C07315=1159.324,218.452,-63.263,-177.799,7.311,148.735
C07316=1159.328,218.203,-63.237,-177.801,7.309,148.735
C07317=1159.332,217.954,-63.212,-177.804,7.306,148.736
C07318=1159.336,217.706,-63.187,-177.807,7.304,148.736
C07319=1159.341,217.457,-63.161,-177.809,7.301,148.736
C07320=1159.346,217.208,-63.137,-177.812,7.300,148.736
C07321=1159.350,216.960,-63.111,-177.815,7.297,148.736
C07322=1159.354,216.711,-63.087,-177.818,7.294,148.737
C07323=1159.359,216.462,-63.061,-177.820,7.292,148.737
C07324=1159.364,216.214,-63.036,-177.823,7.289,148.737
C07325=1159.368,215.965,-63.011,-177.826,7.287,148.737
C07326=1159.372,215.716,-62.987,-177.828,7.284,148.737
C07327=1159.377,215.468,-62.961,-177.831,7.283,148.738
C07328=1159.382,215.219,-62.936,-177.834,7.280,148.738
C07329=1159.386,214.969,-62.911,-177.837,7.277,148.738
C07330=1159.390,214.722,-62.886,-177.839,7.275,148.738
C07331=1159.395,214.472,-62.861,-177.843,7.272,148.738
C07332=1159.400,214.224,-62.836,-177.845,7.270,148.739
C07333=1159.404,213.976,-62.812,-177.848,7.267,148.739
C07334=1159.409,213.726,-62.787,-177.850,7.266,148.739
C07335=1159.413,213.478,-62.761,-177.853,7.263,148.739
C07336=1159.417,213.229,-62.737,-177.856,7.261,148.739
C07337=1159.422,212.980,-62.712,-177.859,7.258,148.739
C07338=1159.427,212.732,-62.687,-177.862,7.255,148.740
C07339=1159.431,212.483,-62.662,-177.864,7.253,148.740
C07340=1159.435,212.234,-62.637,-177.867,7.251,148.740
C07341=1159.440,211.986,-62.612,-177.869,7.248,148.740
C07342=1159.445,211.737,-62.588,-177.873,7.246,148.741
C07343=1159.449,211.488,-62.563,-177.875,7.244,148.741
C07344=1159.454,211.239,-62.538,-177.878,7.241,148.741
C07345=1159.458,210.991,-62.513,-177.880,7.239,148.741
C07346=1159.463,210.742,-62.488,-177.883,7.236,148.741
C07347=1159.467,210.493,-62.464,-177.886,7.234,148.742
C07348=1159.472,210.223,-62.437,-177.889,7.232,148.742
C07349=1159.477,209.952,-62.411,-177.892,7.229,148.742
C07350=1159.482,209.681,-62.383,-177.895,7.226,148.742
C07351=1159.487,209.411,-62.357,-177.898,7.223,148.743
C07352=1159.492,209.163,-62.332,-177.901,7.222,148.743
C07353=1159.496,208.913,-62.308,-177.903,7.219,148.743
C07354=1159.501,208.665,-62.283,-177.906,7.217,148.743
C07355=1159.506,208.416,-62.258,-177.909,7.214,148.743
C07356=1159.510,208.167,-62.234,-177.911,7.212,148.744
C07357=1159.515,207.918,-62.209,-177.914,7.209,148.744
C07358=1159.519,207.670,-62.185,-177.917,7.207,148.744
C07359=1159.524,207.420,-62.160,-177.920,7.205,148.744
C07360=1159.528,207.172,-62.136,-177.922,7.203,148.745
C07361=1159.532,206.924,-62.111,-177.925,7.200,148.745
C07362=1159.537,206.675,-62.086,-177.928,7.198,148.745
C07363=1159.541,206.426,-62.062,-177.931,7.195,148.745
C07364=1159.546,206.178,-62.037,-177.933,7.193,148.746
C07365=1159.551,205.929,-62.014,-177.936,7.190,148.746
C07366=1159.556,205.679,-61.989,-177.939,7.189,148.746
C07367=1159.560,205.431,-61.965,-177.942,7.186,148.746
C07368=1159.565,205.182,-61.940,-177.944,7.184,148.746
C07369=1159.569,204.933,-61.916,-177.947,7.181,148.747
C07370=1159.573,204.684,-61.892,-177.950,7.179,148.747
C07371=1159.578,204.436,-61.867,-177.953,7.177,148.747
C07372=1159.583,204.187,-61.843,-177.955,7.175,148.747
C07373=1159.587,203.938,-61.819,-177.958,7.172,148.748
C07374=1159.592,203.689,-61.794,-177.961,7.170,148.748
C07375=1159.596,203.441,-61.770,-177.964,7.167,148.748
C07376=1159.601,203.192,-61.747,-177.966,7.165,148.748
C07377=1159.605,202.943,-61.721,-177.969,7.163,148.749
C07378=1159.610,202.694,-61.697,-177.971,7.161,148.749
C07379=1159.614,202.446,-61.673,-177.974,7.159,148.749
C07380=1159.619,202.197,-61.649,-177.977,7.156,148.749
C07381=1159.624,201.948,-61.625,-177.980,7.154,148.749
C07382=1159.628,201.699,-61.601,-177.983,7.151,148.750
C07383=1159.633,201.450,-61.576,-177.985,7.149,148.750
C07384=1159.637,201.202,-61.552,-177.988,7.147,148.750
C07385=1159.642,200.953,-61.529,-177.991,7.145,148.750
C07386=1159.646,200.704,-61.505,-177.994,7.142,148.751
C07387=1159.651,200.455,-61.480,-177.996,7.140,148.751
C07388=1159.655,200.207,-61.456,-177.999,7.137,148.751
C07389=1159.660,199.957,-61.432,-178.002,7.136,148.751
C07390=1159.664,199.709,-61.408,-178.005,7.133,148.752
C07391=1159.670,199.460,-61.383,-178.007,7.131,148.752
C07392=1159.674,199.211,-61.360,-178.010,7.129,148.752
C07393=1159.678,198.962,-61.336,-178.013,7.126,148.752
C07394=1159.682,198.714,-61.312,-178.015,7.124,148.753
C07395=1159.687,198.465,-61.288,-178.018,7.122,148.753
C07396=1159.692,198.216,-61.264,-178.021,7.120,148.753
C07397=1159.697,197.967,-61.240,-178.024,7.117,148.753
C07398=1159.701,197.719,-61.216,-178.026,7.115,148.754
C07399=1159.706,197.470,-61.193,-178.029,7.113,148.754
C07400=1159.710,197.221,-61.169,-178.032,7.110,148.754
C07401=1159.714,196.972,-61.144,-178.035,7.109,148.754
C07402=1159.719,196.723,-61.121,-178.037,7.106,148.755
C07403=1159.723,196.475,-61.097,-178.040,7.104,148.755
C07404=1159.729,196.225,-61.073,-178.043,7.101,148.755
C07405=1159.733,195.977,-61.049,-178.046,7.099,148.755
C07406=1159.738,195.728,-61.025,-178.048,7.098,148.756
C07407=1159.742,195.479,-61.001,-178.051,7.095,148.756
C07408=1159.747,195.230,-60.978,-178.054,7.093,148.756
C07409=1159.752,194.981,-60.955,-178.056,7.090,148.756
C07410=1159.756,194.733,-60.931,-178.059,7.088,148.757
C07411=1159.761,194.484,-60.907,-178.062,7.086,148.757
C07412=1159.765,194.235,-60.883,-178.065,7.083,148.757
C07413=1159.770,193.986,-60.860,-178.067,7.082,148.757
C07414=1159.774,193.737,-60.836,-178.071,7.079,148.758
C07415=1159.778,193.488,-60.812,-178.073,7.077,148.758
C07416=1159.783,193.239,-60.789,-178.075,7.075,148.758
C07417=1159.788,192.990,-60.765,-178.078,7.072,148.758
C07418=1159.792,192.742,-60.741,-178.081,7.071,148.759
C07419=1159.797,192.493,-60.718,-178.084,7.068,148.759
C07420=1159.802,192.244,-60.694,-178.086,7.066,148.759
C07421=1159.806,191.995,-60.670,-178.089,7.064,148.760
C07422=1159.811,191.746,-60.647,-178.092,7.062,148.760
C07423=1159.815,191.497,-60.624,-178.095,7.059,148.760
C07424=1159.820,191.249,-60.600,-178.098,7.057,148.760
C07425=1159.824,191.000,-60.576,-178.101,7.055,148.761
C07426=1159.829,190.751,-60.553,-178.103,7.053,148.761
C07427=1159.834,190.502,-60.530,-178.106,7.050,148.761
C07428=1159.839,190.253,-60.506,-178.109,7.049,148.762
C07429=1159.844,190.005,-60.482,-178.111,7.046,148.762
C07430=1159.848,189.756,-60.459,-178.114,7.044,148.762
C07431=1159.853,189.507,-60.436,-178.117,7.042,148.762
C07432=1159.858,189.258,-60.412,-178.120,7.039,148.762
C07433=1159.862,189.009,-60.389,-178.122,7.038,148.763
C07434=1159.866,188.760,-60.366,-178.125,7.036,148.763
C07435=1159.871,188.512,-60.342,-178.128,7.033,148.763
C07436=1159.875,188.263,-60.319,-178.130,7.031,148.764
C07437=1159.880,188.014,-60.295,-178.133,7.029,148.764
C07438=1159.885,187.765,-60.272,-178.136,7.026,148.764
C07439=1159.889,187.516,-60.249,-178.139,7.025,148.764
C07440=1159.893,187.267,-60.226,-178.142,7.022,148.765
C07441=1159.898,187.018,-60.203,-178.144,7.020,148.765
C07442=1159.903,186.769,-60.179,-178.147,7.018,148.765
C07443=1159.908,186.520,-60.156,-178.150,7.016,148.766
C07444=1159.913,186.271,-60.133,-178.152,7.014,148.766
C07445=1159.917,186.023,-60.110,-178.155,7.012,148.766
C07446=1159.922,185.774,-60.087,-178.158,7.009,148.766
C07447=1159.926,185.525,-60.063,-178.160,7.007,148.767
C07448=1159.931,185.276,-60.040,-178.163,7.005,148.767
C07449=1159.936,185.027,-60.017,-178.166,7.003,148.767
C07450=1159.940,184.778,-59.994,-178.169,7.001,148.767
C07451=1159.945,184.530,-59.971,-178.171,6.999,148.768
C07452=1159.950,184.260,-59.946,-178.175,6.996,148.768
C07453=1159.954,183.990,-59.921,-178.178,6.994,148.768
C07454=1159.959,183.720,-59.896,-178.180,6.992,148.769
C07455=1159.964,183.451,-59.870,-178.184,6.989,148.769
C07456=1159.969,183.202,-59.849,-178.186,6.987,148.769
C07457=1159.974,182.953,-59.825,-178.189,6.986,148.770
C07458=1159.979,182.704,-59.802,-178.192,6.983,148.770
C07459=1159.983,182.455,-59.779,-178.194,6.981,148.770
C07460=1159.987,182.206,-59.756,-178.197,6.979,148.771
C07461=1159.992,181.957,-59.732,-178.200,6.977,148.771
C07462=1159.997,181.709,-59.711,-178.203,6.975,148.771
C07463=1160.002,181.460,-59.687,-178.205,6.973,148.771
C07464=1160.006,181.211,-59.664,-178.208,6.970,148.772
C07465=1160.010,180.962,-59.641,-178.211,6.968,148.772
C07466=1160.015,180.713,-59.618,-178.214,6.967,148.772
C07467=1160.020,180.464,-59.596,-178.216,6.964,148.773
C07468=1160.025,180.215,-59.573,-178.219,6.962,148.773
C07469=1160.029,179.966,-59.550,-178.222,6.960,148.773
C07470=1160.034,179.717,-59.527,-178.224,6.958,148.774
C07471=1160.039,179.468,-59.504,-178.227,6.956,148.774
C07472=1160.043,179.220,-59.482,-178.230,6.954,148.774
C07473=1160.048,178.970,-59.459,-178.233,6.952,148.774
C07474=1160.052,178.721,-59.436,-178.236,6.950,148.775
C07475=1160.057,178.473,-59.413,-178.238,6.947,148.775
C07476=1160.062,178.223,-59.391,-178.241,6.946,148.775
C07477=1160.066,177.975,-59.368,-178.243,6.944,148.776
C07478=1160.071,177.726,-59.345,-178.247,6.941,148.776
C07479=1160.076,177.477,-59.323,-178.249,6.939,148.776
C07480=1160.080,177.228,-59.300,-178.252,6.937,148.777
C07481=1160.085,176.979,-59.277,-178.255,6.935,148.777
C07482=1160.090,176.730,-59.254,-178.258,6.933,148.777
C07483=1160.094,176.482,-59.232,-178.260,6.931,148.777
C07484=1160.099,176.232,-59.209,-178.263,6.929,148.778
C07485=1160.103,175.984,-59.187,-178.266,6.927,148.778
C07486=1160.108,175.734,-59.165,-178.268,6.925,148.778
C07487=1160.112,175.485,-59.141,-178.271,6.923,148.779
C07488=1160.117,175.237,-59.120,-178.274,6.920,148.779
C07489=1160.122,174.988,-59.096,-178.277,6.919,148.779
C07490=1160.126,174.738,-59.074,-178.279,6.917,148.780
C07491=1160.132,174.490,-59.051,-178.282,6.915,148.780
C07492=1160.136,174.241,-59.029,-178.285,6.912,148.780
C07493=1160.140,173.991,-59.007,-178.288,6.910,148.781
C07494=1160.145,173.743,-58.984,-178.290,6.909,148.781
C07495=1160.150,173.494,-58.962,-178.293,6.907,148.781
C07496=1160.154,173.245,-58.939,-178.296,6.904,148.782
C07497=1160.159,172.996,-58.917,-178.298,6.902,148.782
C07498=1160.164,172.747,-58.895,-178.301,6.901,148.782
C07499=1160.169,172.498,-58.872,-178.304,6.899,148.782
C07500=1160.173,172.249,-58.850,-178.307,6.896,148.783
C07501=1160.177,172.000,-58.828,-178.310,6.894,148.783
C07502=1160.183,171.751,-58.805,-178.312,6.892,148.783
C07503=1160.187,171.502,-58.783,-178.315,6.891,148.784
C07504=1160.192,171.253,-58.761,-178.318,6.888,148.784
C07505=1160.196,171.004,-58.738,-178.321,6.886,148.784
C07506=1160.201,170.755,-58.716,-178.323,6.885,148.785
C07507=1160.206,170.506,-58.694,-178.325,6.882,148.785
C07508=1160.210,170.257,-58.671,-178.328,6.881,148.785
C07509=1160.215,170.009,-58.649,-178.331,6.878,148.786
C07510=1160.219,169.759,-58.627,-178.334,6.876,148.786
C07511=1160.224,169.511,-58.605,-178.337,6.875,148.786
C07512=1160.229,169.261,-58.583,-178.340,6.873,148.787
C07513=1160.234,169.013,-58.560,-178.342,6.870,148.787
C07514=1160.238,168.764,-58.538,-178.345,6.868,148.787
C07515=1160.243,168.515,-58.517,-178.348,6.866,148.788
C07516=1160.248,168.265,-58.494,-178.350,6.865,148.788
C07517=1160.252,168.016,-58.472,-178.353,6.863,148.788
C07518=1160.257,167.767,-58.450,-178.356,6.860,148.789
C07519=1160.261,167.519,-58.427,-178.359,6.858,148.789
C07520=1160.266,167.270,-58.406,-178.361,6.857,148.789
C07521=1160.271,167.020,-58.383,-178.364,6.855,148.790
C07522=1160.276,166.772,-58.361,-178.367,6.853,148.790
C07523=1160.280,166.522,-58.339,-178.370,6.851,148.790
C07524=1160.285,166.274,-58.318,-178.373,6.849,148.791
C07525=1160.290,166.025,-58.296,-178.375,6.847,148.791
C07526=1160.294,165.776,-58.274,-178.378,6.845,148.791
C07527=1160.299,165.527,-58.252,-178.380,6.843,148.792
C07528=1160.304,165.278,-58.230,-178.384,6.841,148.792
C07529=1160.309,165.029,-58.208,-178.386,6.839,148.792
C07530=1160.313,164.780,-58.186,-178.389,6.837,148.793
C07531=1160.318,164.531,-58.164,-178.392,6.835,148.793
C07532=1160.322,164.282,-58.142,-178.394,6.834,148.793
C07533=1160.327,164.033,-58.120,-178.397,6.831,148.794
C07534=1160.331,163.784,-58.098,-178.400,6.829,148.794
C07535=1160.336,163.535,-58.077,-178.402,6.827,148.794
C07536=1160.341,163.286,-58.055,-178.405,6.826,148.795
C07537=1160.345,163.037,-58.033,-178.408,6.824,148.795
C07538=1160.350,162.788,-58.011,-178.411,6.822,148.795
C07539=1160.355,162.539,-57.989,-178.414,6.819,148.796
C07540=1160.359,162.290,-57.968,-178.417,6.818,148.796
C07541=1160.364,162.041,-57.946,-178.419,6.816,148.796
C07542=1160.370,161.791,-57.924,-178.421,6.814,148.797
C07543=1160.375,161.543,-57.902,-178.424,6.812,148.797
C07544=1160.379,161.293,-57.880,-178.427,6.810,148.797
C07545=1160.384,161.045,-57.859,-178.430,6.808,148.798
C07546=1160.387,160.796,-57.837,-178.433,6.806,148.798
C07547=1160.392,160.547,-57.815,-178.436,6.804,148.799
C07548=1160.397,160.298,-57.794,-178.438,6.803,148.799
C07549=1160.401,160.049,-57.772,-178.441,6.801,148.799
C07550=1160.406,159.800,-57.751,-178.443,6.799,148.799
C07551=1160.411,159.551,-57.729,-178.446,6.796,148.800
C07552=1160.416,159.301,-57.708,-178.449,6.795,148.800
C07553=1160.421,159.053,-57.686,-178.452,6.793,148.801
C07554=1160.426,158.804,-57.664,-178.454,6.791,148.801
C07555=1160.430,158.555,-57.642,-178.457,6.789,148.801
C07556=1160.435,158.285,-57.619,-178.460,6.787,148.802
C07557=1160.440,158.016,-57.596,-178.463,6.785,148.802
C07558=1160.445,157.748,-57.572,-178.466,6.783,148.802
C07559=1160.451,157.479,-57.550,-178.469,6.781,148.803
C07560=1160.455,157.229,-57.528,-178.472,6.779,148.803
C07561=1160.460,156.981,-57.507,-178.475,6.777,148.804
C07562=1160.465,156.732,-57.485,-178.477,6.775,148.804
C07563=1160.469,156.482,-57.464,-178.480,6.774,148.804
C07564=1160.474,156.234,-57.443,-178.483,6.772,148.805
C07565=1160.478,155.985,-57.421,-178.485,6.770,148.805
C07566=1160.483,155.735,-57.400,-178.489,6.768,148.805
C07567=1160.488,155.486,-57.378,-178.491,6.766,148.806
C07568=1160.493,155.237,-57.357,-178.494,6.764,148.806
C07569=1160.497,154.989,-57.336,-178.497,6.762,148.807
C07570=1160.502,154.739,-57.314,-178.499,6.760,148.807
C07571=1160.507,154.490,-57.293,-178.502,6.759,148.807
C07572=1160.512,154.241,-57.272,-178.504,6.757,148.807
C07573=1160.517,153.992,-57.250,-178.507,6.755,148.808
C07574=1160.521,153.743,-57.229,-178.510,6.753,148.808
C07575=1160.525,153.494,-57.208,-178.513,6.751,148.809
C07576=1160.531,153.245,-57.187,-178.516,6.749,148.809
C07577=1160.535,152.996,-57.165,-178.518,6.747,148.809
C07578=1160.540,152.747,-57.145,-178.521,6.746,148.810
C07579=1160.544,152.498,-57.123,-178.524,6.744,148.810
C07580=1160.549,152.249,-57.102,-178.526,6.742,148.810
C07581=1160.554,152.000,-57.080,-178.529,6.740,148.811
C07582=1160.559,151.751,-57.060,-178.532,6.739,148.811
C07583=1160.563,151.501,-57.038,-178.535,6.737,148.812
C07584=1160.568,151.252,-57.017,-178.537,6.735,148.812
C07585=1160.572,151.003,-56.996,-178.541,6.733,148.812
C07586=1160.577,150.755,-56.975,-178.543,6.731,148.813
C07587=1160.583,150.506,-56.954,-178.546,6.729,148.813
C07588=1160.587,150.257,-56.933,-178.549,6.728,148.813
C07589=1160.591,150.007,-56.911,-178.551,6.726,148.814
C07590=1160.596,149.758,-56.890,-178.554,6.724,148.814
C07591=1160.601,149.509,-56.870,-178.557,6.722,148.815
C07592=1160.606,149.260,-56.849,-178.559,6.721,148.815
C07593=1160.611,149.011,-56.827,-178.562,6.719,148.815
C07594=1160.615,148.762,-56.807,-178.564,6.717,148.816
C07595=1160.621,148.513,-56.786,-178.567,6.715,148.816
C07596=1160.625,148.264,-56.764,-178.570,6.713,148.816
C07597=1160.629,148.015,-56.743,-178.573,6.712,148.817
C07598=1160.634,147.765,-56.722,-178.575,6.710,148.817
C07599=1160.639,147.516,-56.702,-178.579,6.707,148.817
C07600=1160.644,147.267,-56.681,-178.581,6.706,148.818
C07601=1160.648,147.019,-56.660,-178.584,6.704,148.818
C07602=1160.653,146.770,-56.639,-178.587,6.702,148.819
C07603=1160.658,146.520,-56.618,-178.589,6.700,148.819
C07604=1160.663,146.271,-56.598,-178.592,6.699,148.819
C07605=1160.668,146.021,-56.576,-178.595,6.697,148.820
C07606=1160.672,145.772,-56.556,-178.597,6.695,148.820
C07607=1160.677,145.523,-56.535,-178.600,6.693,148.821
C07608=1160.681,145.275,-56.514,-178.603,6.692,148.821
C07609=1160.686,145.026,-56.493,-178.606,6.690,148.821
C07610=1160.691,144.777,-56.473,-178.608,6.688,148.822
C07611=1160.696,144.527,-56.452,-178.611,6.686,148.822
C07612=1160.700,144.278,-56.431,-178.614,6.685,148.822
C07613=1160.706,144.029,-56.410,-178.616,6.683,148.823
C07614=1160.710,143.780,-56.390,-178.619,6.681,148.823
C07615=1160.715,143.531,-56.370,-178.622,6.680,148.824
C07616=1160.720,143.282,-56.349,-178.624,6.678,148.824
C07617=1160.724,143.033,-56.328,-178.628,6.676,148.825
C07618=1160.729,142.784,-56.307,-178.630,6.675,148.825
C07619=1160.734,142.535,-56.287,-178.633,6.673,148.825
C07620=1160.739,142.286,-56.266,-178.636,6.671,148.826
C07621=1160.743,142.037,-56.246,-178.638,6.670,148.826
C07622=1160.748,141.788,-56.225,-178.641,6.668,148.827
C07623=1160.753,141.538,-56.204,-178.644,6.666,148.827
C07624=1160.757,141.290,-56.184,-178.647,6.664,148.827
C07625=1160.763,141.040,-56.163,-178.650,6.662,148.828
C07626=1160.767,140.791,-56.143,-178.653,6.660,148.828
C07627=1160.771,140.542,-56.122,-178.655,6.658,148.828
C07628=1160.777,140.293,-56.101,-178.658,6.657,148.829
C07629=1160.781,140.044,-56.082,-178.661,6.655,148.829
C07630=1160.786,139.795,-56.061,-178.663,6.653,148.830
C07631=1160.791,139.545,-56.040,-178.666,6.651,148.830
C07632=1160.795,139.296,-56.020,-178.669,6.650,148.830
C07633=1160.800,139.047,-55.999,-178.671,6.648,148.831
C07634=1160.805,138.798,-55.978,-178.674,6.646,148.831
C07635=1160.809,138.549,-55.958,-178.677,6.644,148.832
C07636=1160.814,138.300,-55.938,-178.680,6.643,148.832
C07637=1160.819,138.050,-55.917,-178.682,6.641,148.832
C07638=1160.824,137.801,-55.897,-178.685,6.639,148.833
C07639=1160.828,137.553,-55.877,-178.688,6.638,148.833
C07640=1160.833,137.303,-55.857,-178.690,6.636,148.833
C07641=1160.838,137.054,-55.836,-178.693,6.635,148.834
C07642=1160.843,136.805,-55.816,-178.696,6.634,148.835
C07643=1160.847,136.556,-55.795,-178.698,6.632,148.835
C07644=1160.852,136.307,-55.776,-178.701,6.630,148.835
C07645=1160.858,136.058,-55.755,-178.704,6.628,148.836
C07646=1160.862,135.809,-55.735,-178.707,6.627,148.836
C07647=1160.867,135.559,-55.715,-178.709,6.625,148.836
C07648=1160.871,135.310,-55.695,-178.712,6.623,148.837
C07649=1160.876,135.061,-55.674,-178.715,6.621,148.837
C07650=1160.881,134.811,-55.654,-178.717,6.620,148.838
C07651=1160.886,134.562,-55.634,-178.720,6.618,148.838
C07652=1160.891,134.314,-55.614,-178.723,6.616,148.838
C07653=1160.895,134.065,-55.594,-178.726,6.615,148.839
C07654=1160.900,133.816,-55.574,-178.728,6.613,148.839
C07655=1160.905,133.566,-55.553,-178.731,6.611,148.840
C07656=1160.910,133.317,-55.533,-178.734,6.610,148.840
C07657=1160.914,133.068,-55.513,-178.737,6.608,148.841
C07658=1160.919,132.818,-55.493,-178.740,6.606,148.841
C07659=1160.924,132.570,-55.473,-178.742,6.605,148.841
C07660=1160.930,132.301,-55.451,-178.745,6.603,148.842
C07661=1160.934,132.032,-55.430,-178.748,6.601,148.842
C07662=1160.939,131.764,-55.408,-178.751,6.600,148.843
C07663=1160.945,131.495,-55.387,-178.754,6.597,148.843
C07664=1160.949,131.247,-55.366,-178.757,6.596,148.844
C07665=1160.954,130.997,-55.347,-178.759,6.595,148.844
C07666=1160.958,130.748,-55.326,-178.762,6.593,148.844
C07667=1160.964,130.499,-55.307,-178.764,6.591,148.845
C07668=1160.968,130.250,-55.287,-178.767,6.589,148.845
C07669=1160.973,130.001,-55.267,-178.770,6.588,148.846
C07670=1160.978,129.751,-55.247,-178.773,6.586,148.846
C07671=1160.982,129.502,-55.227,-178.776,6.585,148.847
C07672=1160.987,129.253,-55.208,-178.778,6.583,148.847
C07673=1160.993,129.004,-55.187,-178.781,6.581,148.847
C07674=1160.997,128.754,-55.167,-178.784,6.579,148.848
C07675=1161.002,128.505,-55.147,-178.787,6.578,148.848
C07676=1161.007,128.257,-55.127,-178.789,6.576,148.849
C07677=1161.012,128.007,-55.108,-178.792,6.574,148.849
C07678=1161.017,127.757,-55.088,-178.795,6.573,148.849
C07679=1161.020,127.509,-55.068,-178.797,6.572,148.850
C07680=1161.026,127.260,-55.049,-178.800,6.570,148.850
C07681=1161.030,127.010,-55.029,-178.803,6.569,148.851
C07682=1161.035,126.761,-55.009,-178.805,6.567,148.851
C07683=1161.040,126.513,-54.990,-178.808,6.565,148.852
C07684=1161.045,126.263,-54.970,-178.811,6.563,148.852
C07685=1161.050,126.013,-54.950,-178.814,6.562,148.852
C07686=1161.054,125.764,-54.930,-178.817,6.560,148.853
C07687=1161.059,125.516,-54.911,-178.819,6.559,148.853
C07688=1161.064,125.266,-54.891,-178.822,6.557,148.854
C07689=1161.069,125.016,-54.871,-178.825,6.555,148.854
C07690=1161.074,124.768,-54.851,-178.827,6.554,148.855
C07691=1161.079,124.519,-54.832,-178.830,6.553,148.855
C07692=1161.083,124.269,-54.813,-178.832,6.551,148.855
C07693=1161.088,124.021,-54.793,-178.835,6.549,148.856
C07694=1161.093,123.771,-54.774,-178.838,6.548,148.856
C07695=1161.098,123.521,-54.754,-178.841,6.546,148.857
C07696=1161.103,123.273,-54.734,-178.844,6.544,148.857
C07697=1161.107,123.024,-54.714,-178.847,6.543,148.858
C07698=1161.112,122.774,-54.695,-178.849,6.541,148.858
C07699=1161.117,122.525,-54.676,-178.851,6.540,148.858
C07700=1161.121,122.276,-54.656,-178.855,6.539,148.859
C07701=1161.126,122.026,-54.637,-178.857,6.537,148.859
C07702=1161.131,121.777,-54.618,-178.860,6.535,148.860
C07703=1161.136,121.528,-54.598,-178.863,6.533,148.860
C07704=1161.141,121.279,-54.579,-178.865,6.532,148.861
C07705=1161.146,121.030,-54.560,-178.868,6.530,148.861
C07706=1161.150,120.780,-54.540,-178.871,6.528,148.861
C07707=1161.155,120.532,-54.520,-178.873,6.528,148.862
C07708=1161.160,120.282,-54.500,-178.876,6.526,148.862
C07709=1161.165,120.034,-54.482,-178.879,6.524,148.863
C07710=1161.169,119.784,-54.462,-178.882,6.523,148.863
C07711=1161.174,119.535,-54.442,-178.884,6.521,148.864
C07712=1161.180,119.285,-54.424,-178.887,6.519,148.864
C07713=1161.184,119.036,-54.405,-178.890,6.518,148.865
C07714=1161.189,118.787,-54.385,-178.892,6.517,148.865
C07715=1161.194,118.537,-54.366,-178.895,6.515,148.865
C07716=1161.199,118.289,-54.347,-178.898,6.514,148.866
C07717=1161.203,118.039,-54.327,-178.900,6.512,148.866
C07718=1161.208,117.790,-54.308,-178.904,6.510,148.867
C07719=1161.213,117.541,-54.289,-178.906,6.509,148.867
C07720=1161.217,117.292,-54.269,-178.909,6.508,148.868
C07721=1161.223,117.043,-54.250,-178.911,6.506,148.868
C07722=1161.227,116.794,-54.231,-178.914,6.504,148.868
C07723=1161.232,116.544,-54.212,-178.917,6.503,148.869
C07724=1161.237,116.294,-54.193,-178.920,6.501,148.870
C07725=1161.242,116.046,-54.174,-178.923,6.500,148.870
C07726=1161.246,115.796,-54.154,-178.925,6.499,148.870
C07727=1161.252,115.548,-54.135,-178.927,6.497,148.871
C07728=1161.256,115.298,-54.116,-178.930,6.495,148.871
C07729=1161.261,115.049,-54.097,-178.933,6.494,148.872
C07730=1161.266,114.799,-54.078,-178.936,6.492,148.872
C07731=1161.271,114.551,-54.059,-178.939,6.491,148.873
C07732=1161.276,114.301,-54.039,-178.941,6.490,148.873
C07733=1161.280,114.052,-54.021,-178.944,6.488,148.873
C07734=1161.285,113.802,-54.002,-178.947,6.487,148.874
C07735=1161.290,113.554,-53.983,-178.950,6.485,148.874
C07736=1161.295,113.304,-53.963,-178.952,6.483,148.875
C07737=1161.300,113.055,-53.945,-178.955,6.481,148.875
C07738=1161.305,112.806,-53.926,-178.957,6.481,148.876
C07739=1161.310,112.557,-53.906,-178.960,6.479,148.876
C07740=1161.314,112.307,-53.888,-178.963,6.477,148.877
C07741=1161.319,112.058,-53.869,-178.966,6.476,148.877
C07742=1161.324,111.809,-53.850,-178.968,6.474,148.878
C07743=1161.329,111.559,-53.831,-178.971,6.473,148.878
C07744=1161.333,111.311,-53.813,-178.974,6.472,148.879
C07745=1161.338,111.061,-53.793,-178.977,6.470,148.879
C07746=1161.343,110.812,-53.775,-178.979,6.468,148.879
C07747=1161.348,110.563,-53.756,-178.982,6.467,148.880
C07748=1161.353,110.313,-53.737,-178.985,6.466,148.880
C07749=1161.358,110.064,-53.718,-178.987,6.464,148.881
C07750=1161.362,109.815,-53.699,-178.990,6.463,148.881
C07751=1161.368,109.565,-53.680,-178.993,6.461,148.882
C07752=1161.372,109.317,-53.662,-178.995,6.460,148.882
C07753=1161.377,109.067,-53.643,-178.998,6.459,148.883
C07754=1161.382,108.818,-53.624,-179.001,6.457,148.883
C07755=1161.387,108.569,-53.606,-179.004,6.455,148.883
C07756=1161.392,108.319,-53.586,-179.006,6.454,148.884
C07757=1161.397,108.070,-53.568,-179.009,6.453,148.885
C07758=1161.401,107.821,-53.549,-179.012,6.451,148.885
C07759=1161.406,107.571,-53.531,-179.014,6.450,148.885
C07760=1161.411,107.323,-53.512,-179.017,6.448,148.886
C07761=1161.416,107.073,-53.493,-179.020,6.447,148.886
C07762=1161.421,106.824,-53.474,-179.022,6.446,148.887
C07763=1161.426,106.575,-53.456,-179.025,6.444,148.887
C07764=1161.431,106.306,-53.436,-179.028,6.442,148.888
C07765=1161.436,106.038,-53.415,-179.031,6.441,148.888
C07766=1161.441,105.770,-53.396,-179.034,6.439,148.889
C07767=1161.447,105.501,-53.376,-179.037,6.438,148.889
C07768=1161.451,105.252,-53.357,-179.040,6.436,148.890
C07769=1161.456,105.003,-53.339,-179.042,6.435,148.890
C07770=1161.462,104.753,-53.320,-179.045,6.434,148.891
C07771=1161.466,104.504,-53.301,-179.048,6.432,148.891
C07772=1161.471,104.255,-53.283,-179.050,6.431,148.892
C07773=1161.475,104.005,-53.265,-179.053,6.430,148.892
C07774=1161.481,103.757,-53.246,-179.056,6.428,148.893
C07775=1161.485,103.507,-53.228,-179.058,6.427,148.893
C07776=1161.490,103.258,-53.210,-179.061,6.425,148.893
C07777=1161.495,103.009,-53.190,-179.063,6.424,148.894
C07778=1161.500,102.759,-53.172,-179.067,6.423,148.895
C07779=1161.505,102.510,-53.154,-179.069,6.421,148.895
C07780=1161.510,102.260,-53.136,-179.072,6.419,148.895
C07781=1161.515,102.012,-53.117,-179.074,6.418,148.896
C07782=1161.519,101.762,-53.098,-179.077,6.417,148.896
C07783=1161.524,101.513,-53.080,-179.080,6.415,148.897
C07784=1161.529,101.263,-53.062,-179.083,6.414,148.897
C07785=1161.534,101.015,-53.044,-179.085,6.413,148.898
C07786=1161.539,100.765,-53.025,-179.088,6.411,148.898
C07787=1161.544,100.515,-53.007,-179.091,6.410,148.899
C07788=1161.548,100.266,-52.989,-179.093,6.409,148.899
C07789=1161.553,100.017,-52.971,-179.096,6.407,148.900
C07790=1161.558,99.768,-52.953,-179.099,6.406,148.900
C07791=1161.563,99.518,-52.933,-179.102,6.404,148.901
C07792=1161.568,99.269,-52.915,-179.104,6.403,148.901
C07793=1161.573,99.020,-52.897,-179.107,6.402,148.902
C07794=1161.578,98.771,-52.879,-179.110,6.400,148.902
C07795=1161.583,98.522,-52.861,-179.112,6.399,148.902
C07796=1161.587,98.272,-52.843,-179.115,6.398,148.903
C07797=1161.592,98.023,-52.825,-179.118,6.396,148.904
C07798=1161.597,97.773,-52.807,-179.120,6.395,148.904
C07799=1161.602,97.524,-52.788,-179.123,6.394,148.904
C07800=1161.607,97.275,-52.770,-179.126,6.392,148.905
C07801=1161.612,97.026,-52.752,-179.129,6.391,148.905
C07802=1161.617,96.776,-52.734,-179.131,6.390,148.906
C07803=1161.621,96.527,-52.715,-179.134,6.388,148.906
C07804=1161.626,96.278,-52.697,-179.137,6.387,148.907
C07805=1161.631,96.029,-52.679,-179.139,6.386,148.907
C07806=1161.636,95.780,-52.662,-179.141,6.384,148.908
C07807=1161.641,95.530,-52.644,-179.145,6.383,148.908
C07808=1161.646,95.281,-52.626,-179.147,6.382,148.909
C07809=1161.650,95.031,-52.608,-179.150,6.380,148.909
C07810=1161.655,94.782,-52.590,-179.153,6.379,148.910
C07811=1161.660,94.532,-52.572,-179.155,6.377,148.910
C07812=1161.665,94.283,-52.554,-179.158,6.376,148.911
C07813=1161.670,94.034,-52.536,-179.161,6.375,148.911
C07814=1161.675,93.785,-52.518,-179.164,6.373,148.912
C07815=1161.680,93.536,-52.500,-179.166,6.372,148.912
C07816=1161.685,93.287,-52.482,-179.169,6.371,148.913
C07817=1161.690,93.037,-52.464,-179.172,6.369,148.913
C07818=1161.695,92.788,-52.446,-179.174,6.368,148.914
C07819=1161.699,92.538,-52.428,-179.177,6.367,148.914
C07820=1161.704,92.288,-52.410,-179.180,6.365,148.915
C07821=1161.709,92.039,-52.393,-179.182,6.364,148.915
C07822=1161.714,91.790,-52.375,-179.185,6.363,148.916
C07823=1161.719,91.541,-52.357,-179.188,6.361,148.916
C07824=1161.724,91.292,-52.339,-179.190,6.361,148.917
C07825=1161.729,91.042,-52.321,-179.193,6.359,148.917
C07826=1161.734,90.793,-52.303,-179.196,6.358,148.918
C07827=1161.739,90.544,-52.285,-179.198,6.357,148.918
C07828=1161.744,90.294,-52.267,-179.201,6.355,148.919
C07829=1161.749,90.045,-52.250,-179.203,6.354,148.919
C07830=1161.753,89.796,-52.233,-179.206,6.353,148.920
C07831=1161.758,89.547,-52.215,-179.209,6.351,148.920
C07832=1161.763,89.297,-52.197,-179.211,6.351,148.921
C07833=1161.768,89.048,-52.179,-179.214,6.349,148.921
C07834=1161.773,88.798,-52.162,-179.217,6.347,148.921
C07835=1161.778,88.549,-52.144,-179.220,6.347,148.922
C07836=1161.783,88.300,-52.126,-179.222,6.345,148.923
C07837=1161.788,88.050,-52.108,-179.225,6.343,148.923
C07838=1161.792,87.801,-52.091,-179.228,6.343,148.924
C07839=1161.798,87.552,-52.074,-179.230,6.341,148.924
C07840=1161.802,87.303,-52.056,-179.233,6.339,148.924
C07841=1161.807,87.053,-52.038,-179.236,6.339,148.925
C07842=1161.813,86.804,-52.020,-179.238,6.337,148.926
C07843=1161.817,86.555,-52.003,-179.241,6.336,148.926
C07844=1161.822,86.306,-51.985,-179.244,6.335,148.927
C07845=1161.827,86.056,-51.968,-179.246,6.333,148.927
C07846=1161.832,85.807,-51.950,-179.249,6.332,148.927
C07847=1161.837,85.557,-51.933,-179.252,6.331,148.928
C07848=1161.841,85.308,-51.915,-179.255,6.329,148.929
C07849=1161.846,85.058,-51.898,-179.257,6.328,148.929
C07850=1161.851,84.809,-51.880,-179.260,6.327,148.930
C07851=1161.856,84.560,-51.862,-179.262,6.326,148.930
C07852=1161.861,84.310,-51.845,-179.265,6.324,148.930
C07853=1161.866,84.061,-51.827,-179.268,6.323,148.931
C07854=1161.871,83.811,-51.810,-179.270,6.322,148.932
C07855=1161.876,83.563,-51.792,-179.273,6.321,148.932
C07856=1161.881,83.313,-51.776,-179.276,6.320,148.933
C07857=1161.886,83.064,-51.758,-179.278,6.318,148.933
C07858=1161.891,82.814,-51.740,-179.281,6.317,148.934
C07859=1161.895,82.565,-51.724,-179.284,6.316,148.934
C07860=1161.900,82.316,-51.706,-179.286,6.314,148.935
C07861=1161.906,82.066,-51.689,-179.289,6.314,148.935
C07862=1161.910,81.817,-51.671,-179.292,6.312,148.936
C07863=1161.915,81.567,-51.654,-179.294,6.311,148.936
C07864=1161.920,81.318,-51.636,-179.297,6.310,148.937
C07865=1161.925,81.069,-51.620,-179.300,6.308,148.937
C07866=1161.930,80.819,-51.602,-179.302,6.308,148.938
C07867=1161.935,80.570,-51.584,-179.305,6.306,148.938
C07868=1161.940,80.302,-51.566,-179.308,6.305,148.939
C07869=1161.946,80.034,-51.548,-179.311,6.304,148.939
C07870=1161.951,79.765,-51.529,-179.314,6.303,148.940
C07871=1161.955,79.497,-51.510,-179.316,6.301,148.940
C07872=1161.961,79.247,-51.493,-179.319,6.299,148.941
C07873=1161.966,78.998,-51.476,-179.322,6.299,148.941
C07874=1161.971,78.749,-51.459,-179.325,6.297,148.942
C07875=1161.976,78.499,-51.442,-179.327,6.297,148.942
C07876=1161.980,78.250,-51.425,-179.330,6.295,148.943
C07877=1161.986,78.000,-51.408,-179.332,6.294,148.943
C07878=1161.990,77.751,-51.390,-179.335,6.293,148.944
C07879=1161.996,77.502,-51.373,-179.338,6.291,148.944
C07880=1162.001,77.252,-51.356,-179.341,6.290,148.945
C07881=1162.005,77.003,-51.340,-179.343,6.289,148.946
C07882=1162.010,76.754,-51.322,-179.346,6.288,148.946
C07883=1162.015,76.504,-51.305,-179.349,6.287,148.947
C07884=1162.020,76.255,-51.288,-179.351,6.286,148.947
C07885=1162.025,76.005,-51.271,-179.354,6.284,148.947
C07886=1162.030,75.756,-51.254,-179.357,6.283,148.948
C07887=1162.034,75.507,-51.237,-179.359,6.282,148.949
C07888=1162.040,75.258,-51.220,-179.362,6.281,148.949
C07889=1162.045,75.008,-51.203,-179.364,6.280,148.950
C07890=1162.050,74.758,-51.186,-179.367,6.278,148.950
C07891=1162.054,74.509,-51.169,-179.370,6.277,148.951
C07892=1162.060,74.260,-51.152,-179.372,6.276,148.951
C07893=1162.065,74.010,-51.136,-179.375,6.275,148.952
C07894=1162.069,73.761,-51.119,-179.378,6.274,148.952
C07895=1162.074,73.512,-51.101,-179.380,6.273,148.953
C07896=1162.079,73.263,-51.085,-179.383,6.271,148.953
C07897=1162.084,73.013,-51.067,-179.385,6.271,148.954
C07898=1162.089,72.764,-51.051,-179.389,6.269,148.954
C07899=1162.094,72.514,-51.033,-179.391,6.268,148.955
C07900=1162.099,72.265,-51.017,-179.393,6.267,148.955
C07901=1162.104,72.016,-51.000,-179.397,6.265,148.956
C07902=1162.109,71.766,-50.983,-179.399,6.264,148.956
C07903=1162.114,71.517,-50.967,-179.402,6.263,148.957
C07904=1162.119,71.267,-50.950,-179.404,6.262,148.957
C07905=1162.124,71.018,-50.933,-179.407,6.261,148.958
C07906=1162.128,70.768,-50.916,-179.410,6.260,148.959
C07907=1162.134,70.519,-50.899,-179.412,6.258,148.959
C07908=1162.138,70.270,-50.883,-179.415,6.258,148.960
C07909=1162.143,70.020,-50.866,-179.418,6.256,148.960
C07910=1162.149,69.771,-50.849,-179.420,6.255,148.960
C07911=1162.153,69.522,-50.832,-179.423,6.254,148.961
C07912=1162.158,69.272,-50.816,-179.425,6.253,148.962
C07913=1162.163,69.023,-50.799,-179.428,6.252,148.962
C07914=1162.168,68.774,-50.782,-179.431,6.251,148.963
C07915=1162.173,68.523,-50.766,-179.434,6.250,148.963
C07916=1162.179,68.274,-50.749,-179.436,6.249,148.964
C07917=1162.183,68.025,-50.733,-179.439,6.247,148.964
C07918=1162.188,67.776,-50.716,-179.441,6.247,148.965
C07919=1162.193,67.527,-50.700,-179.444,6.245,148.965
C07920=1162.198,67.277,-50.682,-179.447,6.244,148.966
C07921=1162.203,67.028,-50.666,-179.449,6.243,148.966
C07922=1162.208,66.778,-50.650,-179.452,6.242,148.967
C07923=1162.212,66.528,-50.634,-179.455,6.241,148.967
C07924=1162.218,66.279,-50.617,-179.457,6.240,148.968
C07925=1162.222,66.030,-50.600,-179.460,6.238,148.969
C07926=1162.227,65.781,-50.584,-179.462,6.238,148.969
C07927=1162.232,65.532,-50.567,-179.465,6.236,148.970
C07928=1162.237,65.281,-50.550,-179.468,6.235,148.970
C07929=1162.243,65.032,-50.534,-179.470,6.234,148.971
C07930=1162.247,64.783,-50.517,-179.473,6.233,148.971
C07931=1162.252,64.534,-50.501,-179.476,6.231,148.972
C07932=1162.257,64.284,-50.485,-179.478,6.231,148.972
C07933=1162.262,64.034,-50.468,-179.481,6.229,148.973
C07934=1162.267,63.785,-50.452,-179.484,6.229,148.973
C07935=1162.272,63.535,-50.436,-179.486,6.227,148.974
C07936=1162.277,63.287,-50.419,-179.489,6.227,148.974
C07937=1162.282,63.037,-50.403,-179.491,6.226,148.975
C07938=1162.287,62.788,-50.386,-179.494,6.224,148.975
C07939=1162.292,62.538,-50.370,-179.497,6.224,148.976
C07940=1162.297,62.289,-50.354,-179.499,6.222,148.976
C07941=1162.302,62.039,-50.338,-179.502,6.221,148.977
C07942=1162.307,61.789,-50.321,-179.505,6.220,148.978
C07943=1162.312,61.541,-50.305,-179.507,6.219,148.978
C07944=1162.316,61.291,-50.289,-179.510,6.218,148.979
C07945=1162.321,61.042,-50.272,-179.512,6.217,148.979
C07946=1162.326,60.792,-50.256,-179.516,6.215,148.980
C07947=1162.332,60.543,-50.240,-179.518,6.214,148.980
C07948=1162.337,60.293,-50.223,-179.520,6.214,148.981
C07949=1162.342,60.044,-50.207,-179.523,6.212,148.981
C07950=1162.346,59.794,-50.191,-179.526,6.212,148.982
C07951=1162.352,59.545,-50.175,-179.528,6.210,148.982
C07952=1162.356,59.295,-50.158,-179.531,6.210,148.983
C07953=1162.361,59.047,-50.142,-179.534,6.208,148.983
C07954=1162.366,58.796,-50.126,-179.536,6.207,148.984
C07955=1162.371,58.548,-50.110,-179.539,6.206,148.985
C07956=1162.377,58.298,-50.094,-179.541,6.205,148.985
C07957=1162.381,58.049,-50.078,-179.544,6.204,148.986
C07958=1162.386,57.799,-50.062,-179.547,6.203,148.986
C07959=1162.391,57.550,-50.045,-179.549,6.202,148.987
C07960=1162.396,57.301,-50.030,-179.552,6.201,148.987
C07961=1162.401,57.050,-50.014,-179.555,6.200,148.988
C07962=1162.406,56.802,-49.997,-179.557,6.198,148.988
C07963=1162.411,56.552,-49.981,-179.560,6.198,148.989
C07964=1162.416,56.303,-49.965,-179.562,6.197,148.989
C07965=1162.421,56.053,-49.950,-179.565,6.196,148.990
C07966=1162.426,55.804,-49.933,-179.568,6.195,148.991
C07967=1162.431,55.554,-49.917,-179.570,6.193,148.991
C07968=1162.436,55.304,-49.901,-179.573,6.193,148.992
C07969=1162.441,55.056,-49.885,-179.576,6.191,148.992
C07970=1162.446,54.805,-49.869,-179.578,6.191,148.993
C07971=1162.451,54.557,-49.853,-179.581,6.190,148.993
C07972=1162.457,54.288,-49.836,-179.584,6.188,148.994
C07973=1162.462,54.020,-49.819,-179.587,6.187,148.995
C07974=1162.467,53.751,-49.801,-179.589,6.186,148.995
C07975=1162.473,53.482,-49.784,-179.592,6.185,148.996
C07976=1162.478,53.233,-49.769,-179.595,6.184,148.996
C07977=1162.483,52.983,-49.752,-179.598,6.183,148.997
C07978=1162.487,52.734,-49.737,-179.600,6.182,148.997
C07979=1162.493,52.485,-49.722,-179.603,6.181,148.998
C07980=1162.497,52.235,-49.706,-179.605,6.180,148.998
C07981=1162.502,51.986,-49.689,-179.608,6.179,148.999
C07982=1162.508,51.736,-49.674,-179.611,6.178,148.999
C07983=1162.513,51.486,-49.658,-179.613,6.177,149.000
C07984=1162.518,51.237,-49.642,-179.615,6.176,149.000
C07985=1162.523,50.988,-49.626,-179.619,6.175,149.001
C07986=1162.527,50.738,-49.611,-179.621,6.174,149.002
C07987=1162.533,50.489,-49.595,-179.623,6.174,149.002
C07988=1162.537,50.239,-49.579,-179.626,6.172,149.003
C07989=1162.543,49.989,-49.563,-179.629,6.171,149.003
C07990=1162.548,49.741,-49.547,-179.632,6.170,149.004
C07991=1162.552,49.492,-49.532,-179.634,6.169,149.004
C07992=1162.557,49.241,-49.516,-179.636,6.168,149.005
C07993=1162.563,48.992,-49.501,-179.640,6.167,149.006
C07994=1162.568,48.743,-49.485,-179.642,6.166,149.006
C07995=1162.573,48.492,-49.469,-179.644,6.165,149.006
C07996=1162.577,48.244,-49.453,-179.647,6.164,149.007
C07997=1162.583,47.995,-49.438,-179.649,6.163,149.008
C07998=1162.587,47.745,-49.422,-179.653,6.162,149.008
C07999=1162.593,47.495,-49.406,-179.655,6.161,149.009
C08000=1162.597,47.246,-49.391,-179.657,6.161,149.009
C08001=1162.603,46.997,-49.376,-179.660,6.159,149.010
C08002=1162.608,46.747,-49.360,-179.663,6.158,149.010
C08003=1162.612,46.497,-49.345,-179.665,6.158,149.011
C08004=1162.618,46.248,-49.329,-179.668,6.156,149.012
C08005=1162.622,45.998,-49.313,-179.670,6.155,149.012
C08006=1162.628,45.749,-49.298,-179.673,6.155,149.013
C08007=1162.632,45.499,-49.283,-179.676,6.153,149.013
C08008=1162.638,45.250,-49.267,-179.678,6.153,149.014
C08009=1162.643,45.000,-49.251,-179.681,6.151,149.014
C08010=1162.647,44.751,-49.236,-179.684,6.151,149.015
C08011=1162.653,44.501,-49.220,-179.686,6.150,149.015
C08012=1162.658,44.252,-49.205,-179.689,6.149,149.016
C08013=1162.663,44.003,-49.190,-179.691,6.148,149.017
C08014=1162.667,43.753,-49.174,-179.694,6.147,149.017
C08015=1162.673,43.503,-49.158,-179.697,6.146,149.018
C08016=1162.677,43.254,-49.143,-179.699,6.145,149.018
C08017=1162.683,43.005,-49.128,-179.701,6.144,149.019
C08018=1162.688,42.756,-49.112,-179.705,6.143,149.019
C08019=1162.692,42.506,-49.097,-179.707,6.142,149.020
C08020=1162.698,42.256,-49.081,-179.709,6.142,149.021
C08021=1162.702,42.007,-49.066,-179.712,6.140,149.021
C08022=1162.708,41.758,-49.051,-179.715,6.139,149.022
C08023=1162.713,41.508,-49.035,-179.717,6.139,149.022
C08024=1162.717,41.258,-49.020,-179.720,6.137,149.023
C08025=1162.723,41.009,-49.005,-179.722,6.136,149.023
C08026=1162.727,40.760,-48.990,-179.725,6.136,149.024
C08027=1162.733,40.510,-48.974,-179.728,6.134,149.024
C08028=1162.738,40.261,-48.959,-179.730,6.134,149.025
C08029=1162.743,40.012,-48.944,-179.733,6.133,149.025
C08030=1162.748,39.761,-48.928,-179.735,6.132,149.026
C08031=1162.753,39.512,-48.913,-179.738,6.131,149.027
C08032=1162.758,39.262,-48.898,-179.741,6.130,149.027
C08033=1162.763,39.013,-48.883,-179.743,6.129,149.028
C08034=1162.768,38.764,-48.867,-179.746,6.128,149.028
C08035=1162.773,38.514,-48.853,-179.748,6.127,149.029
C08036=1162.778,38.265,-48.837,-179.751,6.127,149.029
C08037=1162.783,38.016,-48.822,-179.754,6.125,149.030
C08038=1162.788,37.766,-48.806,-179.756,6.125,149.031
C08039=1162.793,37.516,-48.792,-179.758,6.124,149.031
C08040=1162.798,37.267,-48.777,-179.762,6.123,149.032
C08041=1162.803,37.017,-48.762,-179.764,6.122,149.032
C08042=1162.809,36.767,-48.747,-179.766,6.121,149.033
C08043=1162.813,36.518,-48.732,-179.769,6.120,149.033
C08044=1162.819,36.269,-48.716,-179.772,6.119,149.034
C08045=1162.823,36.020,-48.701,-179.774,6.118,149.034
C08046=1162.829,35.770,-48.686,-179.777,6.118,149.035
C08047=1162.834,35.521,-48.671,-179.780,6.116,149.036
C08048=1162.839,35.271,-48.656,-179.782,6.116,149.036
C08049=1162.843,35.021,-48.641,-179.785,6.115,149.037
C08050=1162.848,34.772,-48.626,-179.787,6.114,149.037
C08051=1162.854,34.522,-48.611,-179.790,6.113,149.038
C08052=1162.858,34.273,-48.596,-179.792,6.112,149.038
C08053=1162.864,34.023,-48.581,-179.795,6.112,149.039
C08054=1162.869,33.774,-48.566,-179.798,6.110,149.040
C08055=1162.874,33.524,-48.551,-179.800,6.110,149.040
C08056=1162.879,33.274,-48.536,-179.802,6.109,149.041
C08057=1162.884,33.025,-48.521,-179.805,6.108,149.041
C08058=1162.889,32.775,-48.507,-179.808,6.107,149.042
C08059=1162.894,32.526,-48.492,-179.810,6.106,149.043
C08060=1162.899,32.277,-48.477,-179.813,6.105,149.043
C08061=1162.904,32.027,-48.462,-179.816,6.104,149.044
C08062=1162.909,31.778,-48.447,-179.818,6.103,149.044
C08063=1162.914,31.528,-48.432,-179.821,6.103,149.045
C08064=1162.919,31.279,-48.417,-179.823,6.102,149.045
C08065=1162.924,31.029,-48.403,-179.826,6.101,149.046
C08066=1162.929,30.780,-48.388,-179.828,6.100,149.046
C08067=1162.935,30.530,-48.373,-179.831,6.099,149.047
C08068=1162.939,30.281,-48.358,-179.833,6.098,149.047
C08069=1162.944,30.031,-48.343,-179.836,6.097,149.048
C08070=1162.950,29.782,-48.328,-179.839,6.097,149.049
C08071=1162.955,29.532,-48.314,-179.841,6.096,149.049
C08072=1162.959,29.282,-48.299,-179.844,6.095,149.050
C08073=1162.964,29.033,-48.284,-179.846,6.094,149.050
C08074=1162.970,28.783,-48.269,-179.849,6.093,149.051
C08075=1162.974,28.534,-48.254,-179.851,6.092,149.052
C08076=1162.980,28.266,-48.239,-179.855,6.091,149.052
C08077=1162.985,27.996,-48.222,-179.857,6.091,149.053
C08078=1162.991,27.727,-48.207,-179.859,6.090,149.053
C08079=1162.996,27.458,-48.192,-179.863,6.088,149.054
C08080=1163.001,27.209,-48.176,-179.865,6.088,149.055
C08081=1163.006,26.959,-48.162,-179.867,6.087,149.055
C08082=1163.012,26.710,-48.148,-179.870,6.087,149.056
C08083=1163.017,26.461,-48.133,-179.873,6.085,149.056
C08084=1163.022,26.211,-48.118,-179.875,6.085,149.057
C08085=1163.027,25.961,-48.104,-179.878,6.084,149.057
C08086=1163.032,25.712,-48.089,-179.880,6.083,149.058
C08087=1163.037,25.462,-48.075,-179.883,6.082,149.059
C08088=1163.042,25.213,-48.060,-179.886,6.081,149.059
C08089=1163.046,24.964,-48.045,-179.888,6.080,149.060
C08090=1163.052,24.714,-48.030,-179.890,6.080,149.060
C08091=1163.057,24.464,-48.016,-179.894,6.079,149.061
C08092=1163.062,24.214,-48.002,-179.896,6.078,149.061
C08093=1163.067,23.966,-47.987,-179.899,6.077,149.062
C08094=1163.072,23.716,-47.973,-179.901,6.076,149.063
C08095=1163.077,23.466,-47.959,-179.903,6.076,149.063
C08096=1163.083,23.216,-47.944,-179.906,6.074,149.064
C08097=1163.088,22.967,-47.929,-179.909,6.074,149.064
C08098=1163.092,22.718,-47.914,-179.911,6.073,149.065
C08099=1163.097,22.468,-47.900,-179.914,6.072,149.066
C08100=1163.102,22.218,-47.886,-179.916,6.072,149.066
C08101=1163.108,21.969,-47.872,-179.919,6.070,149.067
C08102=1163.113,21.719,-47.858,-179.922,6.070,149.067
C08103=1163.118,21.470,-47.843,-179.924,6.069,149.068
C08104=1163.123,21.221,-47.828,-179.926,6.069,149.069
C08105=1163.127,20.971,-47.814,-179.929,6.068,149.069
C08106=1163.133,20.721,-47.799,-179.932,6.066,149.070
C08107=1163.139,20.472,-47.785,-179.934,6.066,149.070
C08108=1163.144,20.222,-47.771,-179.937,6.065,149.071
C08109=1163.149,19.972,-47.757,-179.939,6.064,149.071
C08110=1163.154,19.723,-47.743,-179.941,6.064,149.072
C08111=1163.159,19.473,-47.728,-179.944,6.062,149.072
C08112=1163.163,19.224,-47.713,-179.947,6.062,149.073
C08113=1163.169,18.975,-47.699,-179.950,6.061,149.074
C08114=1163.174,18.725,-47.685,-179.952,6.060,149.074
C08115=1163.179,18.476,-47.671,-179.954,6.060,149.075
C08116=1163.184,18.226,-47.657,-179.957,6.058,149.075
C08117=1163.189,17.976,-47.642,-179.960,6.058,149.076
C08118=1163.194,17.727,-47.628,-179.962,6.057,149.076
C08119=1163.199,17.477,-47.614,-179.965,6.057,149.077
C08120=1163.204,17.228,-47.600,-179.967,6.056,149.078
C08121=1163.209,16.978,-47.586,-179.969,6.055,149.078
C08122=1163.215,16.729,-47.572,-179.972,6.054,149.079
C08123=1163.219,16.479,-47.557,-179.975,6.053,149.079
C08124=1163.224,16.230,-47.543,-179.977,6.053,149.080
C08125=1163.229,15.980,-47.529,-179.980,6.052,149.081
C08126=1163.235,15.731,-47.515,-179.982,6.051,149.081
C08127=1163.240,15.481,-47.501,-179.984,6.051,149.082
C08128=1163.245,15.231,-47.486,-179.988,6.049,149.082
C08129=1163.250,14.982,-47.472,-179.990,6.048,149.083
C08130=1163.255,14.732,-47.459,-179.992,6.048,149.084
C08131=1163.260,14.483,-47.445,-179.995,6.047,149.084
C08132=1163.265,14.233,-47.431,-179.997,6.047,149.085
C08133=1163.270,13.983,-47.417,-180.000,6.046,149.085
C08134=1163.275,13.734,-47.403,179.997,6.045,149.086
C08135=1163.280,13.485,-47.388,179.995,6.044,149.087
C08136=1163.285,13.235,-47.374,179.992,6.043,149.087
C08137=1163.291,12.986,-47.360,179.990,6.043,149.088
C08138=1163.296,12.736,-47.346,179.988,6.042,149.088
C08139=1163.301,12.486,-47.332,179.985,6.042,149.089
C08140=1163.305,12.236,-47.319,179.982,6.040,149.089
C08141=1163.311,11.987,-47.305,179.980,6.039,149.090
C08142=1163.316,11.738,-47.291,179.977,6.039,149.091
C08143=1163.321,11.488,-47.276,179.975,6.038,149.091
C08144=1163.327,11.238,-47.263,179.972,6.038,149.092
C08145=1163.332,10.989,-47.249,179.970,6.037,149.092
C08146=1163.336,10.739,-47.235,179.967,6.036,149.093
C08147=1163.341,10.490,-47.221,179.965,6.036,149.093
C08148=1163.346,10.240,-47.207,179.962,6.034,149.094
C08149=1163.352,9.990,-47.193,179.960,6.033,149.095
C08150=1163.357,9.741,-47.179,179.957,6.033,149.095
C08151=1163.362,9.491,-47.165,179.954,6.033,149.096
C08152=1163.366,9.242,-47.152,179.952,6.032,149.096
C08153=1163.372,8.992,-47.138,179.950,6.031,149.097
C08154=1163.377,8.743,-47.124,179.947,6.030,149.097
C08155=1163.383,8.494,-47.110,179.944,6.029,149.098
C08156=1163.387,8.244,-47.097,179.942,6.028,149.099
C08157=1163.392,7.994,-47.083,179.939,6.028,149.099
C08158=1163.398,7.745,-47.069,179.937,6.027,149.100
C08159=1163.403,7.495,-47.055,179.935,6.027,149.100
C08160=1163.407,7.245,-47.042,179.932,6.026,149.101
C08161=1163.413,6.996,-47.028,179.930,6.025,149.102
C08162=1163.418,6.746,-47.014,179.927,6.025,149.102
C08163=1163.424,6.497,-47.000,179.925,6.024,149.103
C08164=1163.428,6.247,-46.987,179.922,6.023,149.103
C08165=1163.433,5.997,-46.973,179.919,6.022,149.104
C08166=1163.439,5.748,-46.959,179.917,6.021,149.105
C08167=1163.443,5.499,-46.945,179.914,6.021,149.105
C08168=1163.449,5.249,-46.932,179.912,6.020,149.106
C08169=1163.454,4.999,-46.918,179.909,6.020,149.106
C08170=1163.459,4.749,-46.904,179.907,6.019,149.107
C08171=1163.464,4.500,-46.891,179.905,6.018,149.108
C08172=1163.469,4.250,-46.878,179.902,6.018,149.108
C08173=1163.474,4.001,-46.864,179.899,6.016,149.109
C08174=1163.479,3.752,-46.850,179.896,6.016,149.109
C08175=1163.485,3.502,-46.837,179.894,6.015,149.110
C08176=1163.490,3.252,-46.823,179.892,6.015,149.111
C08177=1163.495,3.003,-46.810,179.889,6.014,149.111
C08178=1163.500,2.753,-46.796,179.887,6.013,149.112
C08179=1163.504,2.503,-46.783,179.885,6.012,149.112
C08180=1163.510,2.235,-46.768,179.882,6.012,149.113
C08181=1163.516,1.965,-46.753,179.879,6.011,149.114
C08182=1163.521,1.695,-46.739,179.876,6.010,149.114
C08183=1163.527,1.426,-46.724,179.874,6.009,149.115
C08184=1163.532,1.176,-46.711,179.871,6.009,149.115
C08185=1163.537,0.927,-46.697,179.869,6.009,149.116
C08186=1163.542,0.677,-46.684,179.866,6.008,149.117
C08187=1163.547,0.428,-46.670,179.864,6.007,149.117
C08188=1163.552,0.178,-46.657,179.862,6.006,149.118
C08189=1163.557,-0.071,-46.643,179.858,6.005,149.118
C08190=1163.563,-0.321,-46.630,179.856,6.004,149.119
C08191=1163.567,-0.571,-46.617,179.854,6.004,149.120
C08192=1163.573,-0.820,-46.603,179.851,6.003,149.120
C08193=1163.577,-1.070,-46.590,179.849,6.003,149.121
C08194=1163.583,-1.319,-46.576,179.846,6.002,149.121
C08195=1163.588,-1.568,-46.564,179.844,6.001,149.122
C08196=1163.593,-1.819,-46.550,179.841,6.001,149.123
C08197=1163.598,-2.067,-46.537,179.839,6.000,149.123
C08198=1163.603,-2.318,-46.523,179.836,6.000,149.124
C08199=1163.609,-2.567,-46.511,179.834,5.999,149.124
C08200=1163.614,-2.817,-46.496,179.832,5.998,149.125
C08201=1163.619,-3.066,-46.484,179.829,5.998,149.126
C08202=1163.624,-3.316,-46.470,179.827,5.997,149.126
C08203=1163.629,-3.565,-46.457,179.824,5.997,149.127
C08204=1163.634,-3.816,-46.443,179.821,5.995,149.127
C08205=1163.639,-4.065,-46.431,179.819,5.995,149.128
C08206=1163.645,-4.314,-46.417,179.816,5.994,149.129
C08207=1163.649,-4.564,-46.404,179.814,5.993,149.129
C08208=1163.655,-4.813,-46.391,179.811,5.993,149.130
C08209=1163.660,-5.064,-46.378,179.809,5.992,149.130
C08210=1163.665,-5.313,-46.364,179.806,5.992,149.131
C08211=1163.670,-5.563,-46.351,179.804,5.991,149.131
C08212=1163.676,-5.812,-46.338,179.801,5.990,149.132
C08213=1163.681,-6.061,-46.325,179.799,5.990,149.133
C08214=1163.685,-6.312,-46.312,179.797,5.989,149.133
C08215=1163.691,-6.561,-46.299,179.794,5.989,149.134
C08216=1163.695,-6.811,-46.285,179.792,5.988,149.134
C08217=1163.701,-7.060,-46.272,179.789,5.987,149.135
C08218=1163.706,-7.309,-46.259,179.787,5.987,149.135
C08219=1163.711,-7.559,-46.246,179.784,5.986,149.136
C08220=1163.717,-7.809,-46.233,179.782,5.986,149.137
C08221=1163.721,-8.058,-46.220,179.780,5.985,149.137
C08222=1163.727,-8.308,-46.206,179.777,5.984,149.138
C08223=1163.732,-8.557,-46.194,179.775,5.984,149.138
C08224=1163.736,-8.807,-46.181,179.772,5.983,149.139
C08225=1163.742,-9.057,-46.167,179.770,5.982,149.140
C08226=1163.747,-9.306,-46.155,179.767,5.982,149.140
C08227=1163.752,-9.556,-46.142,179.765,5.981,149.141
C08228=1163.758,-9.806,-46.129,179.762,5.981,149.141
C08229=1163.763,-10.055,-46.116,179.760,5.980,149.142
C08230=1163.767,-10.305,-46.102,179.758,5.979,149.143
C08231=1163.773,-10.554,-46.089,179.755,5.979,149.143
C08232=1163.778,-10.804,-46.077,179.753,5.978,149.144
C08233=1163.783,-11.054,-46.064,179.750,5.978,149.144
C08234=1163.788,-11.303,-46.050,179.747,5.977,149.145
C08235=1163.794,-11.553,-46.038,179.745,5.976,149.146
C08236=1163.798,-11.803,-46.025,179.742,5.975,149.146
C08237=1163.803,-12.052,-46.012,179.740,5.974,149.147
C08238=1163.809,-12.302,-45.999,179.737,5.974,149.147
C08239=1163.814,-12.552,-45.986,179.735,5.973,149.148
C08240=1163.819,-12.801,-45.974,179.732,5.973,149.149
C08241=1163.825,-13.051,-45.960,179.730,5.972,149.149
C08242=1163.830,-13.300,-45.948,179.727,5.971,149.150
C08243=1163.834,-13.550,-45.935,179.725,5.971,149.150
C08244=1163.839,-13.799,-45.922,179.723,5.970,149.151
C08245=1163.844,-14.049,-45.910,179.720,5.970,149.152
C08246=1163.850,-14.299,-45.896,179.718,5.969,149.152
C08247=1163.855,-14.548,-45.883,179.715,5.968,149.153
C08248=1163.860,-14.798,-45.871,179.712,5.968,149.154
C08249=1163.865,-15.048,-45.859,179.711,5.968,149.154
C08250=1163.871,-15.298,-45.845,179.708,5.967,149.155
C08251=1163.876,-15.547,-45.833,179.706,5.967,149.155
C08252=1163.881,-15.796,-45.820,179.703,5.966,149.156
C08253=1163.886,-16.046,-45.808,179.701,5.965,149.156
C08254=1163.891,-16.296,-45.795,179.699,5.965,149.157
C08255=1163.896,-16.545,-45.781,179.696,5.964,149.158
C08256=1163.902,-16.795,-45.769,179.694,5.964,149.158
C08257=1163.907,-17.045,-45.757,179.691,5.963,149.159
C08258=1163.911,-17.295,-45.744,179.689,5.962,149.159
C08259=1163.917,-17.544,-45.731,179.686,5.962,149.160
C08260=1163.922,-17.793,-45.719,179.684,5.961,149.160
C08261=1163.928,-18.043,-45.706,179.681,5.961,149.161
C08262=1163.933,-18.292,-45.693,179.679,5.960,149.162
C08263=1163.938,-18.543,-45.681,179.677,5.959,149.162
C08264=1163.943,-18.792,-45.668,179.674,5.959,149.163
C08265=1163.948,-19.042,-45.656,179.672,5.958,149.164
C08266=1163.953,-19.291,-45.643,179.669,5.958,149.164
C08267=1163.958,-19.540,-45.630,179.667,5.957,149.165
C08268=1163.964,-19.791,-45.617,179.664,5.957,149.165
C08269=1163.969,-20.040,-45.605,179.662,5.956,149.166
C08270=1163.974,-20.290,-45.592,179.659,5.955,149.167
C08271=1163.979,-20.539,-45.580,179.657,5.955,149.167
C08272=1163.984,-20.789,-45.568,179.655,5.954,149.168
C08273=1163.989,-21.039,-45.555,179.652,5.954,149.168
C08274=1163.994,-21.288,-45.542,179.650,5.953,149.169
C08275=1163.999,-21.538,-45.530,179.647,5.952,149.170
C08276=1164.005,-21.788,-45.518,179.644,5.952,149.170
C08277=1164.010,-22.037,-45.505,179.642,5.951,149.171
C08278=1164.015,-22.286,-45.493,179.640,5.951,149.171
C08279=1164.020,-22.536,-45.481,179.637,5.950,149.172
C08280=1164.025,-22.786,-45.468,179.635,5.949,149.173
C08281=1164.031,-23.036,-45.454,179.633,5.949,149.173
C08282=1164.036,-23.286,-45.443,179.630,5.949,149.174
C08283=1164.041,-23.535,-45.430,179.628,5.948,149.174
C08284=1164.047,-23.805,-45.417,179.626,5.948,149.175
C08285=1164.052,-24.074,-45.404,179.622,5.946,149.176
C08286=1164.058,-24.345,-45.390,179.620,5.946,149.176
C08287=1164.063,-24.615,-45.376,179.617,5.946,149.177
C08288=1164.068,-24.864,-45.364,179.615,5.945,149.177
C08289=1164.074,-25.114,-45.352,179.612,5.944,149.178
C08290=1164.079,-25.363,-45.339,179.610,5.944,149.179
C08291=1164.084,-25.613,-45.327,179.607,5.943,149.179
C08292=1164.089,-25.863,-45.315,179.606,5.943,149.180
C08293=1164.095,-26.113,-45.303,179.603,5.943,149.181
C08294=1164.100,-26.362,-45.290,179.600,5.942,149.181
C08295=1164.105,-26.611,-45.278,179.598,5.941,149.182
C08296=1164.109,-26.862,-45.266,179.596,5.941,149.182
C08297=1164.114,-27.111,-45.254,179.593,5.940,149.183
C08298=1164.120,-27.361,-45.242,179.591,5.940,149.184
C08299=1164.125,-27.610,-45.229,179.589,5.939,149.184
C08300=1164.130,-27.860,-45.217,179.586,5.939,149.185
C08301=1164.135,-28.109,-45.205,179.583,5.938,149.185
C08302=1164.141,-28.359,-45.193,179.581,5.937,149.186
C08303=1164.146,-28.609,-45.180,179.578,5.937,149.187
C08304=1164.151,-28.859,-45.168,179.576,5.936,149.187
C08305=1164.157,-29.108,-45.156,179.574,5.936,149.188
C08306=1164.162,-29.358,-45.144,179.572,5.936,149.188
C08307=1164.167,-29.607,-45.131,179.569,5.935,149.189
C08308=1164.172,-29.857,-45.120,179.567,5.934,149.189
C08309=1164.177,-30.107,-45.108,179.564,5.934,149.190
C08310=1164.182,-30.356,-45.095,179.562,5.934,149.191
C08311=1164.188,-30.606,-45.083,179.560,5.933,149.191
C08312=1164.193,-30.855,-45.071,179.557,5.932,149.192
C08313=1164.198,-31.105,-45.059,179.555,5.931,149.192
C08314=1164.203,-31.355,-45.046,179.552,5.931,149.193
C08315=1164.208,-31.604,-45.035,179.550,5.930,149.194
C08316=1164.214,-31.854,-45.023,179.548,5.931,149.194
C08317=1164.219,-32.103,-45.011,179.545,5.930,149.195
C08318=1164.224,-32.353,-44.999,179.543,5.929,149.195
C08319=1164.230,-32.603,-44.987,179.540,5.929,149.196
C08320=1164.235,-32.853,-44.974,179.538,5.928,149.197
C08321=1164.239,-33.102,-44.963,179.535,5.928,149.197
C08322=1164.244,-33.352,-44.950,179.533,5.927,149.198
C08323=1164.250,-33.602,-44.938,179.531,5.927,149.198
C08324=1164.255,-33.851,-44.927,179.528,5.926,149.199
C08325=1164.261,-34.101,-44.915,179.526,5.926,149.200
C08326=1164.265,-34.350,-44.903,179.524,5.926,149.200
C08327=1164.271,-34.600,-44.891,179.522,5.925,149.201
C08328=1164.276,-34.850,-44.879,179.519,5.924,149.202
C08329=1164.281,-35.100,-44.866,179.517,5.924,149.202
C08330=1164.286,-35.349,-44.855,179.514,5.923,149.203
C08331=1164.291,-35.599,-44.843,179.512,5.922,149.203
C08332=1164.297,-35.849,-44.831,179.509,5.922,149.204
C08333=1164.302,-36.098,-44.819,179.507,5.922,149.205
C08334=1164.306,-36.348,-44.807,179.505,5.922,149.205
C08335=1164.312,-36.598,-44.795,179.502,5.921,149.206
C08336=1164.317,-36.848,-44.784,179.500,5.920,149.206
C08337=1164.322,-37.097,-44.771,179.497,5.920,149.207
C08338=1164.327,-37.347,-44.760,179.495,5.919,149.207
C08339=1164.333,-37.597,-44.748,179.493,5.919,149.208
C08340=1164.339,-37.846,-44.736,179.490,5.918,149.209
C08341=1164.344,-38.096,-44.724,179.488,5.917,149.209
C08342=1164.348,-38.345,-44.712,179.486,5.918,149.210
C08343=1164.354,-38.595,-44.701,179.483,5.917,149.210
C08344=1164.359,-38.845,-44.689,179.481,5.917,149.211
C08345=1164.364,-39.094,-44.677,179.479,5.916,149.212
C08346=1164.369,-39.344,-44.665,179.476,5.915,149.212
C08347=1164.375,-39.594,-44.654,179.474,5.915,149.213
C08348=1164.379,-39.843,-44.642,179.471,5.914,149.214
C08349=1164.385,-40.093,-44.630,179.470,5.914,149.214
C08350=1164.391,-40.343,-44.618,179.467,5.914,149.215
C08351=1164.395,-40.592,-44.607,179.464,5.913,149.215
C08352=1164.401,-40.842,-44.595,179.462,5.912,149.216
C08353=1164.406,-41.092,-44.583,179.459,5.912,149.217
C08354=1164.411,-41.342,-44.572,179.457,5.911,149.217
C08355=1164.416,-41.592,-44.560,179.455,5.911,149.218
C08356=1164.421,-41.841,-44.549,179.453,5.911,149.218
C08357=1164.427,-42.091,-44.537,179.450,5.910,149.219
C08358=1164.433,-42.340,-44.525,179.448,5.910,149.219
C08359=1164.437,-42.589,-44.513,179.445,5.909,149.220
C08360=1164.442,-42.839,-44.501,179.443,5.908,149.221
C08361=1164.447,-43.089,-44.490,179.441,5.908,149.221
C08362=1164.452,-43.339,-44.478,179.439,5.908,149.222
C08363=1164.458,-43.589,-44.466,179.436,5.908,149.222
C08364=1164.463,-43.838,-44.455,179.434,5.907,149.223
C08365=1164.469,-44.088,-44.443,179.431,5.906,149.224
C08366=1164.473,-44.337,-44.432,179.429,5.906,149.224
C08367=1164.479,-44.587,-44.420,179.427,5.905,149.225
C08368=1164.483,-44.837,-44.409,179.425,5.905,149.225
C08369=1164.489,-45.087,-44.397,179.422,5.905,149.226
C08370=1164.494,-45.336,-44.386,179.420,5.904,149.227
C08371=1164.500,-45.586,-44.374,179.417,5.904,149.227
C08372=1164.505,-45.836,-44.362,179.415,5.903,149.228
C08373=1164.510,-46.086,-44.352,179.412,5.903,149.229
C08374=1164.515,-46.336,-44.340,179.411,5.903,149.229
C08375=1164.521,-46.585,-44.329,179.408,5.902,149.230
C08376=1164.526,-46.835,-44.317,179.406,5.901,149.230
C08377=1164.531,-47.084,-44.306,179.403,5.901,149.231
C08378=1164.536,-47.334,-44.294,179.401,5.900,149.231
C08379=1164.542,-47.583,-44.283,179.398,5.900,149.232
C08380=1164.547,-47.833,-44.271,179.397,5.900,149.233
C08381=1164.552,-48.083,-44.260,179.394,5.899,149.233
C08382=1164.557,-48.333,-44.248,179.392,5.899,149.234
C08383=1164.562,-48.582,-44.237,179.389,5.898,149.234
C08384=1164.568,-48.832,-44.226,179.386,5.898,149.235
C08385=1164.573,-49.082,-44.215,179.385,5.898,149.236
C08386=1164.578,-49.331,-44.203,179.382,5.897,149.236
C08387=1164.583,-49.581,-44.191,179.380,5.897,149.237
C08388=1164.589,-49.852,-44.180,179.377,5.896,149.237
C08389=1164.594,-50.122,-44.167,179.375,5.896,149.238
C08390=1164.601,-50.392,-44.155,179.372,5.895,149.239
C08391=1164.606,-50.663,-44.143,179.370,5.894,149.239
C08392=1164.611,-50.913,-44.131,179.367,5.894,149.240
C08393=1164.616,-51.162,-44.120,179.365,5.893,149.241
C08394=1164.622,-51.412,-44.108,179.363,5.894,149.241
C08395=1164.627,-51.662,-44.098,179.361,5.893,149.242
C08396=1164.632,-51.912,-44.086,179.358,5.892,149.242
C08397=1164.637,-52.161,-44.075,179.356,5.892,149.243
C08398=1164.642,-52.410,-44.064,179.353,5.891,149.244
C08399=1164.648,-52.661,-44.052,179.352,5.891,149.244
C08400=1164.653,-52.910,-44.042,179.349,5.891,149.245
C08401=1164.658,-53.160,-44.030,179.346,5.890,149.246
C08402=1164.663,-53.409,-44.018,179.344,5.890,149.246
C08403=1164.668,-53.660,-44.008,179.342,5.890,149.247
C08404=1164.674,-53.909,-43.996,179.340,5.889,149.247
C08405=1164.679,-54.159,-43.985,179.337,5.889,149.248
C08406=1164.684,-54.409,-43.974,179.335,5.888,149.248
C08407=1164.690,-54.658,-43.963,179.332,5.888,149.249
C08408=1164.695,-54.908,-43.952,179.331,5.888,149.250
C08409=1164.699,-55.157,-43.940,179.328,5.887,149.250
C08410=1164.705,-55.407,-43.930,179.326,5.886,149.251
C08411=1164.710,-55.657,-43.918,179.323,5.886,149.251
C08412=1164.715,-55.906,-43.907,179.321,5.885,149.252
C08413=1164.721,-56.156,-43.897,179.319,5.886,149.253
C08414=1164.726,-56.406,-43.885,179.317,5.885,149.253
C08415=1164.731,-56.656,-43.874,179.314,5.884,149.254
C08416=1164.736,-56.905,-43.863,179.312,5.884,149.254
C08417=1164.742,-57.155,-43.851,179.310,5.884,149.255
C08418=1164.747,-57.405,-43.841,179.307,5.884,149.256
C08419=1164.752,-57.654,-43.830,179.305,5.883,149.256
C08420=1164.757,-57.904,-43.819,179.302,5.882,149.257
C08421=1164.763,-58.154,-43.808,179.300,5.882,149.257
C08422=1164.768,-58.403,-43.797,179.298,5.882,149.258
C08423=1164.773,-58.653,-43.786,179.296,5.881,149.259
C08424=1164.778,-58.902,-43.775,179.293,5.881,149.259
C08425=1164.784,-59.153,-43.764,179.291,5.880,149.260
C08426=1164.789,-59.403,-43.753,179.289,5.880,149.260
C08427=1164.794,-59.652,-43.742,179.287,5.880,149.261
C08428=1164.799,-59.902,-43.731,179.284,5.879,149.262
C08429=1164.805,-60.151,-43.720,179.282,5.878,149.262
C08430=1164.810,-60.401,-43.709,179.280,5.879,149.263
C08431=1164.815,-60.651,-43.698,179.278,5.878,149.263
C08432=1164.820,-60.900,-43.688,179.275,5.878,149.264
C08433=1164.825,-61.150,-43.676,179.273,5.877,149.264
C08434=1164.831,-61.400,-43.665,179.271,5.877,149.265
C08435=1164.836,-61.650,-43.654,179.268,5.876,149.266
C08436=1164.841,-61.900,-43.644,179.266,5.876,149.266
C08437=1164.846,-62.149,-43.633,179.264,5.875,149.267
C08438=1164.851,-62.399,-43.622,179.262,5.876,149.267
C08439=1164.857,-62.648,-43.612,179.259,5.875,149.268
C08440=1164.862,-62.898,-43.600,179.257,5.874,149.269
C08441=1164.868,-63.148,-43.590,179.255,5.874,149.269
C08442=1164.873,-63.398,-43.578,179.252,5.874,149.270
C08443=1164.878,-63.647,-43.568,179.250,5.873,149.270
C08444=1164.883,-63.897,-43.557,179.248,5.873,149.271
C08445=1164.888,-64.147,-43.546,179.245,5.872,149.272
C08446=1164.893,-64.397,-43.536,179.243,5.872,149.272
C08447=1164.899,-64.646,-43.524,179.241,5.872,149.273
C08448=1164.904,-64.896,-43.514,179.238,5.871,149.273
C08449=1164.909,-65.146,-43.503,179.236,5.870,149.274
C08450=1164.915,-65.395,-43.493,179.234,5.871,149.275
C08451=1164.920,-65.645,-43.482,179.232,5.870,149.275
C08452=1164.925,-65.894,-43.471,179.229,5.870,149.276
C08453=1164.930,-66.145,-43.461,179.227,5.869,149.276
C08454=1164.936,-66.394,-43.450,179.225,5.869,149.277
C08455=1164.940,-66.644,-43.439,179.223,5.868,149.277
C08456=1164.947,-66.894,-43.428,179.220,5.868,149.278
C08457=1164.952,-67.144,-43.418,179.219,5.868,149.279
C08458=1164.957,-67.393,-43.407,179.216,5.868,149.279
C08459=1164.962,-67.643,-43.396,179.214,5.867,149.280
C08460=1164.968,-67.893,-43.386,179.211,5.866,149.281
C08461=1164.972,-68.142,-43.375,179.210,5.866,149.281
C08462=1164.978,-68.392,-43.364,179.207,5.866,149.282
C08463=1164.983,-68.642,-43.354,179.205,5.865,149.282
C08464=1164.988,-68.892,-43.344,179.202,5.865,149.283
C08465=1164.993,-69.141,-43.332,179.200,5.865,149.283
C08466=1164.999,-69.391,-43.322,179.198,5.864,149.284
C08467=1165.004,-69.641,-43.312,179.196,5.864,149.285
C08468=1165.009,-69.890,-43.301,179.193,5.864,149.285
C08469=1165.015,-70.139,-43.290,179.191,5.863,149.286
C08470=1165.020,-70.390,-43.280,179.189,5.863,149.286
C08471=1165.025,-70.639,-43.270,179.186,5.862,149.287
C08472=1165.030,-70.889,-43.259,179.184,5.863,149.288
C08473=1165.036,-71.138,-43.248,179.182,5.862,149.288
C08474=1165.041,-71.389,-43.238,179.179,5.861,149.289
C08475=1165.046,-71.638,-43.227,179.178,5.861,149.289
C08476=1165.051,-71.888,-43.217,179.175,5.861,149.290
C08477=1165.057,-72.138,-43.207,179.173,5.860,149.291
C08478=1165.062,-72.387,-43.196,179.171,5.861,149.291
C08479=1165.067,-72.637,-43.185,179.169,5.860,149.292
C08480=1165.073,-72.887,-43.175,179.166,5.859,149.292
C08481=1165.078,-73.137,-43.164,179.164,5.859,149.293
C08482=1165.083,-73.386,-43.154,179.162,5.859,149.294
C08483=1165.089,-73.636,-43.144,179.160,5.858,149.294
C08484=1165.094,-73.886,-43.133,179.157,5.858,149.295
C08485=1165.099,-74.135,-43.122,179.155,5.858,149.295
C08486=1165.104,-74.385,-43.112,179.153,5.857,149.296
C08487=1165.110,-74.635,-43.102,179.150,5.857,149.296
C08488=1165.115,-74.884,-43.091,179.148,5.857,149.297
C08489=1165.120,-75.135,-43.081,179.146,5.856,149.298
C08490=1165.126,-75.384,-43.071,179.144,5.856,149.298
C08491=1165.131,-75.634,-43.060,179.142,5.856,149.299
C08492=1165.137,-75.905,-43.050,179.139,5.855,149.300
C08493=1165.143,-76.177,-43.038,179.137,5.855,149.300
C08494=1165.147,-76.447,-43.026,179.134,5.854,149.301
C08495=1165.154,-76.718,-43.015,179.132,5.854,149.301
C08496=1165.159,-76.969,-43.005,179.130,5.853,149.302
C08497=1165.164,-77.218,-42.995,179.127,5.854,149.303
C08498=1165.169,-77.467,-42.985,179.125,5.853,149.303
C08499=1165.174,-77.718,-42.974,179.123,5.852,149.304
C08500=1165.180,-77.967,-42.964,179.121,5.852,149.304
C08501=1165.186,-78.217,-42.954,179.118,5.852,149.305
C08502=1165.191,-78.467,-42.943,179.116,5.851,149.306
C08503=1165.196,-78.716,-42.933,179.114,5.852,149.306
C08504=1165.202,-78.966,-42.923,179.112,5.851,149.307
C08505=1165.206,-79.216,-42.913,179.109,5.850,149.307
C08506=1165.212,-79.465,-42.903,179.108,5.850,149.308
C08507=1165.217,-79.715,-42.892,179.105,5.850,149.308
C08508=1165.222,-79.965,-42.882,179.103,5.849,149.309
C08509=1165.228,-80.215,-42.872,179.101,5.849,149.310
C08510=1165.233,-80.464,-42.862,179.098,5.849,149.310
C08511=1165.238,-80.715,-42.852,179.096,5.848,149.311
C08512=1165.244,-80.964,-42.842,179.094,5.849,149.311
C08513=1165.249,-81.214,-42.832,179.092,5.848,149.312
C08514=1165.255,-81.464,-42.821,179.089,5.847,149.313
C08515=1165.259,-81.713,-42.812,179.088,5.847,149.313
C08516=1165.265,-81.963,-42.801,179.085,5.847,149.314
C08517=1165.270,-82.213,-42.791,179.083,5.846,149.314
C08518=1165.275,-82.463,-42.781,179.081,5.846,149.315
C08519=1165.281,-82.712,-42.770,179.079,5.846,149.316
C08520=1165.286,-82.962,-42.761,179.076,5.845,149.316
C08521=1165.292,-83.212,-42.751,179.074,5.845,149.317
C08522=1165.297,-83.462,-42.741,179.072,5.845,149.317
C08523=1165.302,-83.712,-42.730,179.070,5.844,149.318
C08524=1165.307,-83.961,-42.721,179.068,5.844,149.318
C08525=1165.312,-84.211,-42.710,179.065,5.844,149.319
C08526=1165.318,-84.461,-42.700,179.064,5.844,149.320
C08527=1165.323,-84.710,-42.690,179.061,5.844,149.320
C08528=1165.328,-84.960,-42.681,179.059,5.843,149.321
C08529=1165.333,-85.210,-42.670,179.057,5.843,149.321
C08530=1165.339,-85.460,-42.660,179.055,5.842,149.322
C08531=1165.344,-85.709,-42.651,179.052,5.842,149.322
C08532=1165.350,-85.958,-42.640,179.050,5.842,149.323
C08533=1165.355,-86.209,-42.630,179.048,5.841,149.324
C08534=1165.360,-86.459,-42.621,179.045,5.841,149.324
C08535=1165.365,-86.708,-42.611,179.044,5.841,149.325
C08536=1165.371,-86.958,-42.600,179.041,5.840,149.326
C08537=1165.376,-87.207,-42.591,179.039,5.840,149.326
C08538=1165.381,-87.458,-42.581,179.037,5.840,149.327
C08539=1165.387,-87.707,-42.571,179.035,5.839,149.327
C08540=1165.392,-87.957,-42.561,179.033,5.839,149.328
C08541=1165.397,-88.206,-42.551,179.030,5.839,149.328
C08542=1165.402,-88.457,-42.541,179.028,5.838,149.329
C08543=1165.407,-88.706,-42.531,179.026,5.839,149.330
C08544=1165.413,-88.956,-42.521,179.024,5.838,149.330
C08545=1165.418,-89.206,-42.512,179.022,5.837,149.331
C08546=1165.424,-89.455,-42.502,179.020,5.837,149.331
C08547=1165.429,-89.705,-42.492,179.017,5.837,149.332
C08548=1165.434,-89.955,-42.483,179.015,5.836,149.332
C08549=1165.439,-90.205,-42.472,179.013,5.836,149.333
C08550=1165.445,-90.454,-42.462,179.011,5.836,149.334
C08551=1165.450,-90.704,-42.453,179.009,5.836,149.334
C08552=1165.456,-90.954,-42.443,179.007,5.835,149.335
C08553=1165.460,-91.204,-42.433,179.004,5.835,149.335
C08554=1165.466,-91.454,-42.424,179.002,5.835,149.336
C08555=1165.472,-91.703,-42.413,179.000,5.834,149.337
C08556=1165.476,-91.953,-42.404,178.998,5.834,149.337
C08557=1165.482,-92.203,-42.394,178.996,5.834,149.338
C08558=1165.487,-92.452,-42.385,178.993,5.833,149.338
C08559=1165.492,-92.702,-42.374,178.992,5.833,149.339
C08560=1165.497,-92.952,-42.365,178.989,5.833,149.339
C08561=1165.503,-93.202,-42.355,178.987,5.832,149.340
C08562=1165.508,-93.451,-42.346,178.985,5.833,149.341
C08563=1165.514,-93.701,-42.336,178.983,5.832,149.341
C08564=1165.519,-93.951,-42.326,178.981,5.832,149.342
C08565=1165.524,-94.200,-42.317,178.978,5.831,149.342
C08566=1165.529,-94.451,-42.306,178.976,5.831,149.343
C08567=1165.535,-94.700,-42.297,178.974,5.831,149.343
C08568=1165.540,-94.950,-42.287,178.972,5.830,149.344
C08569=1165.545,-95.200,-42.278,178.970,5.830,149.344
C08570=1165.551,-95.449,-42.268,178.968,5.830,149.345
C08571=1165.556,-95.699,-42.259,178.965,5.829,149.346
C08572=1165.562,-95.949,-42.249,178.963,5.830,149.346
C08573=1165.567,-96.199,-42.240,178.961,5.829,149.347
C08574=1165.573,-96.448,-42.230,178.958,5.828,149.348
C08575=1165.577,-96.699,-42.221,178.957,5.828,149.348
C08576=1165.583,-96.948,-42.210,178.955,5.828,149.349
C08577=1165.588,-97.198,-42.201,178.953,5.828,149.349
C08578=1165.593,-97.448,-42.191,178.950,5.827,149.350
C08579=1165.599,-97.698,-42.182,178.948,5.826,149.350
C08580=1165.604,-97.947,-42.172,178.946,5.827,149.351
C08581=1165.609,-98.197,-42.163,178.944,5.826,149.351
C08582=1165.615,-98.446,-42.153,178.942,5.827,149.352
C08583=1165.620,-98.696,-42.144,178.940,5.826,149.353
C08584=1165.625,-98.946,-42.135,178.938,5.826,149.353
C08585=1165.631,-99.196,-42.125,178.935,5.825,149.354
C08586=1165.636,-99.445,-42.115,178.933,5.825,149.354
C08587=1165.642,-99.695,-42.106,178.931,5.825,149.355
C08588=1165.647,-99.945,-42.097,178.929,5.824,149.355
C08589=1165.652,-100.195,-42.087,178.927,5.824,149.356
C08590=1165.657,-100.445,-42.078,178.925,5.824,149.357
C08591=1165.662,-100.694,-42.068,178.922,5.823,149.357
C08592=1165.668,-100.944,-42.058,178.920,5.824,149.358
C08593=1165.673,-101.194,-42.050,178.918,5.823,149.358
C08594=1165.679,-101.444,-42.039,178.917,5.823,149.359
C08595=1165.684,-101.694,-42.030,178.914,5.822,149.360
C08596=1165.689,-101.966,-42.020,178.912,5.822,149.360
C08597=1165.695,-102.237,-42.010,178.910,5.822,149.361
C08598=1165.702,-102.509,-42.000,178.907,5.821,149.361
C08599=1165.707,-102.781,-41.989,178.905,5.821,149.362
C08600=1165.712,-103.031,-41.980,178.903,5.821,149.362
C08601=1165.718,-103.280,-41.970,178.900,5.821,149.363
C08602=1165.723,-103.530,-41.961,178.898,5.820,149.364
C08603=1165.728,-103.780,-41.952,178.896,5.820,149.364
C08604=1165.734,-104.030,-41.943,178.894,5.819,149.365
C08605=1165.739,-104.280,-41.933,178.892,5.819,149.365
C08606=1165.744,-104.529,-41.924,178.890,5.819,149.366
C08607=1165.750,-104.780,-41.915,178.888,5.819,149.367
C08608=1165.755,-105.029,-41.905,178.886,5.818,149.367
C08609=1165.760,-105.279,-41.896,178.884,5.819,149.368
C08610=1165.766,-105.529,-41.887,178.882,5.818,149.368
C08611=1165.771,-105.779,-41.878,178.879,5.817,149.369
C08612=1165.776,-106.028,-41.868,178.877,5.818,149.369
C08613=1165.781,-106.278,-41.860,178.875,5.817,149.370
C08614=1165.787,-106.528,-41.850,178.873,5.817,149.371
C08615=1165.792,-106.778,-41.841,178.871,5.817,149.371
C08616=1165.797,-107.027,-41.831,178.869,5.817,149.372
C08617=1165.803,-107.277,-41.822,178.867,5.816,149.372
C08618=1165.808,-107.527,-41.813,178.864,5.815,149.373
C08619=1165.813,-107.777,-41.804,178.863,5.815,149.373
C08620=1165.818,-108.026,-41.795,178.860,5.815,149.374
C08621=1165.824,-108.276,-41.785,178.859,5.815,149.374
C08622=1165.829,-108.526,-41.776,178.856,5.814,149.375
C08623=1165.834,-108.776,-41.767,178.854,5.815,149.376
C08624=1165.840,-109.025,-41.759,178.852,5.814,149.376
C08625=1165.846,-109.275,-41.749,178.851,5.814,149.377
C08626=1165.851,-109.524,-41.740,178.848,5.814,149.377
C08627=1165.856,-109.774,-41.731,178.846,5.813,149.378
C08628=1165.861,-110.024,-41.722,178.844,5.813,149.378
C08629=1165.867,-110.274,-41.712,178.841,5.813,149.379
C08630=1165.872,-110.524,-41.703,178.840,5.813,149.380
C08631=1165.877,-110.774,-41.695,178.837,5.812,149.380
C08632=1165.882,-111.023,-41.685,178.836,5.812,149.381
C08633=1165.888,-111.273,-41.675,178.833,5.811,149.381
C08634=1165.893,-111.523,-41.667,178.831,5.812,149.382
C08635=1165.899,-111.773,-41.658,178.829,5.811,149.382
C08636=1165.904,-112.022,-41.649,178.827,5.811,149.383
C08637=1165.909,-112.272,-41.640,178.825,5.811,149.384
C08638=1165.915,-112.522,-41.631,178.823,5.810,149.384
C08639=1165.921,-112.772,-41.622,178.821,5.810,149.385
C08640=1165.926,-113.022,-41.613,178.818,5.810,149.385
C08641=1165.931,-113.272,-41.604,178.817,5.810,149.386
C08642=1165.936,-113.522,-41.595,178.815,5.809,149.386
C08643=1165.941,-113.772,-41.586,178.813,5.809,149.387
C08644=1165.947,-114.020,-41.576,178.810,5.809,149.387
C08645=1165.953,-114.270,-41.568,178.809,5.809,149.388
C08646=1165.958,-114.520,-41.559,178.806,5.808,149.388
C08647=1165.963,-114.770,-41.550,178.804,5.808,149.389
C08648=1165.968,-115.020,-41.541,178.802,5.808,149.390
C08649=1165.973,-115.270,-41.532,178.801,5.808,149.390
C08650=1165.978,-115.519,-41.523,178.798,5.807,149.391
C08651=1165.985,-115.769,-41.514,178.796,5.807,149.391
C08652=1165.990,-116.019,-41.505,178.794,5.806,149.392
C08653=1165.995,-116.269,-41.496,178.792,5.807,149.393
C08654=1166.000,-116.519,-41.487,178.790,5.806,149.393
C08655=1166.006,-116.768,-41.478,178.788,5.805,149.394
C08656=1166.011,-117.018,-41.469,178.786,5.806,149.394
C08657=1166.016,-117.268,-41.461,178.783,5.805,149.395
C08658=1166.022,-117.517,-41.452,178.782,5.805,149.395
C08659=1166.027,-117.768,-41.444,178.779,5.805,149.396
C08660=1166.033,-118.018,-41.434,178.777,5.805,149.396
C08661=1166.038,-118.268,-41.425,178.775,5.804,149.397
C08662=1166.043,-118.518,-41.417,178.774,5.804,149.397
C08663=1166.049,-118.767,-41.408,178.771,5.804,149.398
C08664=1166.054,-119.017,-41.399,178.769,5.804,149.399
C08665=1166.059,-119.266,-41.390,178.767,5.803,149.399
C08666=1166.065,-119.516,-41.381,178.765,5.803,149.400
C08667=1166.070,-119.766,-41.372,178.763,5.803,149.400
C08668=1166.076,-120.015,-41.364,178.761,5.803,149.401
C08669=1166.081,-120.265,-41.355,178.759,5.802,149.401
C08670=1166.086,-120.515,-41.346,178.757,5.802,149.402
C08671=1166.091,-120.765,-41.338,178.755,5.801,149.402
C08672=1166.097,-121.015,-41.329,178.753,5.801,149.403
C08673=1166.102,-121.264,-41.320,178.751,5.801,149.404
C08674=1166.107,-121.514,-41.312,178.749,5.801,149.404
C08675=1166.113,-121.764,-41.303,178.747,5.800,149.405
C08676=1166.118,-122.014,-41.294,178.745,5.801,149.405
C08677=1166.123,-122.264,-41.285,178.743,5.800,149.406
C08678=1166.129,-122.514,-41.277,178.741,5.800,149.406
C08679=1166.134,-122.763,-41.268,178.739,5.799,149.407
C08680=1166.139,-123.013,-41.259,178.737,5.800,149.407
C08681=1166.145,-123.263,-41.250,178.734,5.799,149.408
C08682=1166.150,-123.512,-41.242,178.733,5.799,149.408
C08683=1166.155,-123.762,-41.233,178.731,5.798,149.409
C08684=1166.161,-124.013,-41.225,178.729,5.799,149.410
C08685=1166.166,-124.262,-41.216,178.726,5.798,149.410
C08686=1166.172,-124.512,-41.207,178.725,5.798,149.411
C08687=1166.177,-124.761,-41.198,178.722,5.798,149.411
C08688=1166.183,-125.012,-41.190,178.721,5.798,149.412
C08689=1166.188,-125.262,-41.181,178.718,5.797,149.412
C08690=1166.193,-125.511,-41.173,178.717,5.797,149.413
C08691=1166.199,-125.761,-41.164,178.714,5.797,149.414
C08692=1166.204,-126.011,-41.156,178.712,5.797,149.414
C08693=1166.210,-126.260,-41.147,178.710,5.796,149.415
C08694=1166.215,-126.510,-41.138,178.709,5.796,149.415
C08695=1166.220,-126.760,-41.129,178.706,5.795,149.416
C08696=1166.225,-127.010,-41.122,178.704,5.796,149.416
C08697=1166.231,-127.259,-41.113,178.702,5.795,149.417
C08698=1166.236,-127.509,-41.104,178.701,5.795,149.417
C08699=1166.241,-127.760,-41.096,178.698,5.794,149.418
C08700=1165.820,-127.770,-41.137,178.695,5.798,149.420
C08701=1165.815,-127.520,-41.146,178.697,5.798,149.419
C08702=1165.810,-127.271,-41.154,178.699,5.799,149.419
C08703=1165.804,-127.021,-41.163,178.700,5.799,149.418
C08704=1165.799,-126.771,-41.171,178.703,5.800,149.418
C08705=1165.793,-126.521,-41.180,178.705,5.799,149.417
C08706=1165.788,-126.271,-41.189,178.706,5.799,149.416
C08707=1165.782,-126.022,-41.197,178.709,5.800,149.416
C08708=1165.777,-125.772,-41.206,178.710,5.800,149.415
C08709=1165.772,-125.522,-41.215,178.713,5.800,149.415
C08710=1165.767,-125.273,-41.222,178.714,5.800,149.414
C08711=1165.761,-125.023,-41.231,178.717,5.801,149.414
C08712=1165.756,-124.773,-41.240,178.719,5.800,149.413
C08713=1165.751,-124.523,-41.248,178.721,5.801,149.412
C08714=1165.745,-124.274,-41.257,178.722,5.801,149.412
C08715=1165.740,-124.024,-41.266,178.725,5.802,149.412
C08716=1165.735,-123.773,-41.274,178.727,5.801,149.411
C08717=1165.729,-123.523,-41.283,178.729,5.802,149.410
C08718=1165.724,-123.274,-41.291,178.731,5.802,149.410
C08719=1165.719,-123.024,-41.300,178.733,5.803,149.409
C08720=1165.713,-122.775,-41.309,178.735,5.803,149.409
C08721=1165.708,-122.524,-41.317,178.737,5.803,149.408
C08722=1165.702,-122.275,-41.326,178.739,5.803,149.408
C08723=1165.697,-122.025,-41.335,178.741,5.804,149.407
C08724=1165.692,-121.775,-41.344,178.743,5.804,149.406
C08725=1165.687,-121.525,-41.353,178.745,5.804,149.406
C08726=1165.681,-121.276,-41.361,178.747,5.804,149.405
C08727=1165.675,-121.026,-41.369,178.749,5.805,149.405
C08728=1165.670,-120.776,-41.378,178.751,5.805,149.404
C08729=1165.665,-120.526,-41.387,178.753,5.805,149.404
C08730=1165.660,-120.276,-41.396,178.755,5.806,149.403
C08731=1165.654,-120.027,-41.405,178.757,5.806,149.403
C08732=1165.649,-119.777,-41.414,178.760,5.807,149.402
C08733=1165.644,-119.527,-41.422,178.761,5.807,149.402
C08734=1165.639,-119.278,-41.431,178.764,5.807,149.401
C08735=1165.633,-119.028,-41.440,178.766,5.807,149.400
C08736=1165.627,-118.778,-41.449,178.768,5.808,149.400
C08737=1165.622,-118.528,-41.458,178.770,5.807,149.399
C08738=1165.616,-118.278,-41.466,178.772,5.808,149.399
C08739=1165.611,-118.028,-41.475,178.774,5.808,149.398
C08740=1165.606,-117.778,-41.484,178.776,5.809,149.398
C08741=1165.601,-117.528,-41.493,178.778,5.808,149.397
C08742=1165.595,-117.279,-41.502,178.780,5.809,149.397
C08743=1165.590,-117.029,-41.511,178.782,5.809,149.396
C08744=1165.585,-116.780,-41.519,178.784,5.809,149.395
C08745=1165.580,-116.530,-41.528,178.786,5.809,149.395
C08746=1165.574,-116.280,-41.537,178.788,5.810,149.394
C08747=1165.569,-116.030,-41.547,178.790,5.810,149.394
C08748=1165.563,-115.781,-41.555,178.792,5.810,149.393
C08749=1165.558,-115.531,-41.564,178.794,5.810,149.393
C08750=1165.552,-115.281,-41.573,178.796,5.811,149.392
C08751=1165.547,-115.031,-41.582,178.798,5.811,149.391
C08752=1165.542,-114.781,-41.591,178.800,5.812,149.391
C08753=1165.537,-114.531,-41.600,178.803,5.812,149.390
C08754=1165.530,-114.282,-41.609,178.805,5.812,149.390
C08755=1165.525,-114.032,-41.618,178.807,5.813,149.389
C08756=1165.520,-113.782,-41.627,178.809,5.813,149.389
C08757=1165.515,-113.532,-41.636,178.811,5.813,149.388
C08758=1165.510,-113.282,-41.644,178.813,5.813,149.388
C08759=1165.505,-113.033,-41.653,178.815,5.814,149.387
C08760=1165.499,-112.782,-41.663,178.817,5.813,149.386
C08761=1165.494,-112.533,-41.672,178.819,5.814,149.386
C08762=1165.488,-112.284,-41.681,178.821,5.814,149.385
C08763=1165.483,-112.034,-41.690,178.824,5.814,149.385
C08764=1165.478,-111.784,-41.699,178.825,5.814,149.384
C08765=1165.473,-111.534,-41.708,178.827,5.815,149.384
C08766=1165.467,-111.284,-41.717,178.830,5.815,149.383
C08767=1165.461,-111.034,-41.726,178.832,5.815,149.383
C08768=1165.456,-110.785,-41.735,178.834,5.816,149.382
C08769=1165.451,-110.535,-41.744,178.836,5.816,149.381
C08770=1165.445,-110.285,-41.753,178.838,5.817,149.381
C08771=1165.440,-110.035,-41.763,178.840,5.817,149.380
C08772=1165.435,-109.786,-41.772,178.842,5.817,149.380
C08773=1165.429,-109.536,-41.780,178.844,5.817,149.379
C08774=1165.424,-109.287,-41.789,178.846,5.818,149.379
C08775=1165.418,-109.036,-41.799,178.848,5.817,149.378
C08776=1165.413,-108.786,-41.808,178.850,5.818,149.377
C08777=1165.408,-108.537,-41.817,178.853,5.819,149.377
C08778=1165.403,-108.287,-41.826,178.855,5.818,149.376
C08779=1165.397,-108.037,-41.836,178.857,5.819,149.376
C08780=1165.392,-107.787,-41.845,178.859,5.819,149.375
C08781=1165.387,-107.538,-41.854,178.861,5.819,149.375
C08782=1165.381,-107.288,-41.864,178.863,5.819,149.374
C08783=1165.376,-107.038,-41.873,178.865,5.820,149.374
C08784=1165.371,-106.788,-41.882,178.867,5.820,149.373
C08785=1165.366,-106.538,-41.890,178.869,5.821,149.372
C08786=1165.360,-106.289,-41.901,178.872,5.821,149.372
C08787=1165.355,-106.039,-41.910,178.874,5.821,149.371
C08788=1165.350,-105.789,-41.918,178.876,5.822,149.371
C08789=1165.344,-105.539,-41.928,178.878,5.821,149.370
C08790=1165.339,-105.290,-41.938,178.880,5.822,149.370
C08791=1165.334,-105.040,-41.946,178.882,5.822,149.369
C08792=1165.328,-104.790,-41.956,178.884,5.822,149.368
C08793=1165.323,-104.540,-41.965,178.886,5.823,149.368
C08794=1165.318,-104.291,-41.974,178.888,5.823,149.367
C08795=1165.312,-104.041,-41.984,178.891,5.823,149.367
C08796=1165.307,-103.791,-41.993,178.892,5.823,149.366
C08797=1165.302,-103.541,-42.002,178.895,5.824,149.366
C08798=1165.296,-103.291,-42.012,178.897,5.824,149.365
C08799=1165.291,-103.041,-42.021,178.899,5.825,149.365
C08800=1165.286,-102.792,-42.030,178.901,5.825,149.364
C08801=1165.281,-102.520,-42.041,178.903,5.825,149.363
C08802=1165.274,-102.248,-42.050,178.906,5.825,149.363
C08803=1165.268,-101.976,-42.061,178.908,5.826,149.362
C08804=1165.263,-101.704,-42.071,178.910,5.826,149.361
C08805=1165.258,-101.455,-42.080,178.912,5.826,149.361
C08806=1165.252,-101.205,-42.090,178.915,5.827,149.360
C08807=1165.247,-100.955,-42.099,178.916,5.827,149.360
C08808=1165.241,-100.706,-42.109,178.919,5.828,149.359
C08809=1165.236,-100.456,-42.118,178.921,5.827,149.359
C08810=1165.231,-100.206,-42.128,178.923,5.828,149.358
C08811=1165.225,-99.956,-42.137,178.926,5.828,149.357
C08812=1165.220,-99.706,-42.146,178.927,5.828,149.357
C08813=1165.214,-99.457,-42.156,178.929,5.829,149.356
C08814=1165.209,-99.207,-42.165,178.931,5.829,149.356
C08815=1165.204,-98.957,-42.175,178.934,5.829,149.355
C08816=1165.199,-98.707,-42.185,178.936,5.829,149.354
C08817=1165.194,-98.458,-42.194,178.938,5.830,149.354
C08818=1165.188,-98.208,-42.204,178.940,5.831,149.353
C08819=1165.183,-97.958,-42.213,178.942,5.830,149.353
C08820=1165.177,-97.708,-42.223,178.944,5.831,149.352
C08821=1165.172,-97.458,-42.232,178.946,5.831,149.352
C08822=1165.167,-97.209,-42.242,178.949,5.831,149.351
C08823=1165.162,-96.959,-42.251,178.951,5.832,149.351
C08824=1165.156,-96.709,-42.261,178.953,5.832,149.350
C08825=1165.151,-96.459,-42.270,178.955,5.832,149.349
C08826=1165.145,-96.210,-42.280,178.957,5.832,149.349
C08827=1165.140,-95.960,-42.289,178.959,5.833,149.348
C08828=1165.135,-95.710,-42.300,178.962,5.834,149.348
C08829=1165.130,-95.460,-42.308,178.964,5.833,149.347
C08830=1165.124,-95.210,-42.319,178.966,5.834,149.347
C08831=1165.119,-94.961,-42.328,178.967,5.834,149.346
C08832=1165.113,-94.711,-42.338,178.970,5.834,149.345
C08833=1165.109,-94.462,-42.347,178.972,5.835,149.345
C08834=1165.103,-94.212,-42.357,178.974,5.835,149.344
C08835=1165.098,-93.962,-42.367,178.977,5.835,149.344
C08836=1165.092,-93.712,-42.376,178.979,5.836,149.343
C08837=1165.088,-93.462,-42.386,178.981,5.836,149.342
C08838=1165.082,-93.212,-42.395,178.983,5.837,149.342
C08839=1165.076,-92.963,-42.406,178.985,5.836,149.341
C08840=1165.071,-92.713,-42.415,178.987,5.837,149.341
C08841=1165.065,-92.463,-42.425,178.990,5.837,149.340
C08842=1165.061,-92.214,-42.434,178.992,5.837,149.340
C08843=1165.055,-91.964,-42.444,178.994,5.838,149.339
C08844=1165.050,-91.714,-42.454,178.996,5.838,149.338
C08845=1165.045,-91.464,-42.464,178.998,5.838,149.338
C08846=1165.039,-91.214,-42.474,179.001,5.839,149.337
C08847=1165.034,-90.965,-42.483,179.002,5.839,149.337
C08848=1165.028,-90.715,-42.493,179.005,5.840,149.336
C08849=1165.023,-90.466,-42.502,179.007,5.840,149.335
C08850=1165.018,-90.215,-42.513,179.009,5.840,149.335
C08851=1165.013,-89.966,-42.523,179.012,5.840,149.334
C08852=1165.008,-89.716,-42.532,179.013,5.840,149.334
C08853=1165.002,-89.466,-42.542,179.016,5.841,149.333
C08854=1164.997,-89.217,-42.552,179.018,5.841,149.333
C08855=1164.992,-88.966,-42.562,179.020,5.841,149.332
C08856=1164.986,-88.717,-42.572,179.022,5.842,149.331
C08857=1164.981,-88.468,-42.581,179.024,5.843,149.331
C08858=1164.976,-88.218,-42.592,179.027,5.842,149.330
C08859=1164.970,-87.968,-42.601,179.029,5.843,149.330
C08860=1164.966,-87.718,-42.611,179.031,5.843,149.329
C08861=1164.960,-87.468,-42.621,179.033,5.843,149.329
C08862=1164.954,-87.219,-42.632,179.035,5.844,149.328
C08863=1164.949,-86.969,-42.640,179.037,5.844,149.327
C08864=1164.944,-86.719,-42.651,179.039,5.844,149.327
C08865=1164.939,-86.469,-42.661,179.042,5.845,149.326
C08866=1164.934,-86.220,-42.671,179.044,5.845,149.326
C08867=1164.928,-85.970,-42.680,179.046,5.845,149.325
C08868=1164.922,-85.720,-42.691,179.049,5.846,149.325
C08869=1164.918,-85.470,-42.701,179.051,5.846,149.324
C08870=1164.912,-85.221,-42.711,179.053,5.846,149.323
C08871=1164.907,-84.971,-42.721,179.055,5.847,149.323
C08872=1164.902,-84.721,-42.730,179.057,5.847,149.322
C08873=1164.897,-84.471,-42.740,179.059,5.847,149.322
C08874=1164.891,-84.222,-42.751,179.062,5.848,149.321
C08875=1164.885,-83.972,-42.761,179.064,5.848,149.320
C08876=1164.881,-83.722,-42.771,179.066,5.848,149.320
C08877=1164.876,-83.473,-42.781,179.068,5.849,149.319
C08878=1164.870,-83.223,-42.791,179.070,5.849,149.319
C08879=1164.864,-82.973,-42.801,179.073,5.849,149.318
C08880=1164.860,-82.723,-42.811,179.074,5.849,149.318
C08881=1164.854,-82.473,-42.821,179.077,5.850,149.317
C08882=1164.849,-82.224,-42.831,179.079,5.851,149.316
C08883=1164.843,-81.974,-42.841,179.081,5.850,149.316
C08884=1164.839,-81.724,-42.851,179.083,5.851,149.315
C08885=1164.833,-81.475,-42.862,179.086,5.851,149.314
C08886=1164.828,-81.225,-42.872,179.088,5.851,149.314
C08887=1164.823,-80.975,-42.882,179.090,5.852,149.313
C08888=1164.817,-80.725,-42.893,179.093,5.852,149.313
C08889=1164.812,-80.476,-42.901,179.094,5.852,149.312
C08890=1164.807,-80.225,-42.912,179.097,5.853,149.312
C08891=1164.801,-79.976,-42.922,179.099,5.854,149.311
C08892=1164.796,-79.726,-42.932,179.101,5.853,149.310
C08893=1164.791,-79.476,-42.943,179.103,5.854,149.310
C08894=1164.786,-79.227,-42.953,179.106,5.854,149.309
C08895=1164.780,-78.977,-42.963,179.108,5.854,149.309
C08896=1164.775,-78.727,-42.973,179.110,5.855,149.308
C08897=1164.770,-78.477,-42.984,179.112,5.856,149.308
C08898=1164.764,-78.228,-42.994,179.115,5.856,149.307
C08899=1164.759,-77.978,-43.004,179.117,5.856,149.306
C08900=1164.753,-77.728,-43.015,179.119,5.856,149.306
C08901=1164.748,-77.479,-43.024,179.122,5.857,149.305
C08902=1164.743,-77.229,-43.035,179.123,5.857,149.305
C08903=1164.738,-76.979,-43.045,179.126,5.858,149.304
C08904=1164.732,-76.730,-43.055,179.128,5.858,149.304
C08905=1164.726,-76.458,-43.067,179.130,5.858,149.303
C08906=1164.721,-76.187,-43.078,179.133,5.858,149.302
C08907=1164.715,-75.916,-43.090,179.135,5.859,149.302
C08908=1164.710,-75.645,-43.101,179.138,5.859,149.301
C08909=1164.704,-75.396,-43.111,179.140,5.860,149.300
C08910=1164.699,-75.145,-43.121,179.142,5.860,149.300
C08911=1164.694,-74.896,-43.132,179.145,5.860,149.299
C08912=1164.688,-74.646,-43.142,179.147,5.861,149.299
C08913=1164.683,-74.396,-43.152,179.149,5.861,149.298
C08914=1164.677,-74.146,-43.162,179.151,5.861,149.297
C08915=1164.672,-73.896,-43.173,179.153,5.862,149.297
C08916=1164.667,-73.647,-43.184,179.155,5.862,149.296
C08917=1164.661,-73.398,-43.194,179.157,5.863,149.296
C08918=1164.656,-73.147,-43.205,179.160,5.863,149.295
C08919=1164.651,-72.898,-43.215,179.162,5.864,149.294
C08920=1164.647,-72.648,-43.225,179.164,5.863,149.294
C08921=1164.641,-72.398,-43.235,179.167,5.864,149.293
C08922=1164.635,-72.149,-43.245,179.169,5.865,149.293
C08923=1164.631,-71.899,-43.257,179.171,5.865,149.292
C08924=1164.625,-71.650,-43.267,179.174,5.865,149.291
C08925=1164.620,-71.400,-43.277,179.176,5.866,149.291
C08926=1164.615,-71.150,-43.288,179.178,5.866,149.290
C08927=1164.610,-70.900,-43.298,179.180,5.866,149.290
C08928=1164.604,-70.651,-43.309,179.183,5.866,149.289
C08929=1164.599,-70.401,-43.320,179.185,5.867,149.289
C08930=1164.594,-70.151,-43.330,179.187,5.867,149.288
C08931=1164.588,-69.901,-43.340,179.189,5.868,149.287
C08932=1164.583,-69.651,-43.351,179.192,5.868,149.287
C08933=1164.578,-69.402,-43.362,179.194,5.869,149.286
C08934=1164.572,-69.152,-43.373,179.196,5.868,149.285
C08935=1164.566,-68.902,-43.383,179.198,5.869,149.285
C08936=1164.562,-68.653,-43.394,179.201,5.870,149.284
C08937=1164.556,-68.403,-43.405,179.202,5.870,149.284
C08938=1164.551,-68.153,-43.415,179.205,5.870,149.283
C08939=1164.546,-67.903,-43.425,179.207,5.871,149.283
C08940=1164.541,-67.654,-43.437,179.210,5.871,149.282
C08941=1164.535,-67.404,-43.447,179.212,5.871,149.281
C08942=1164.530,-67.154,-43.457,179.214,5.872,149.281
C08943=1164.525,-66.905,-43.468,179.216,5.872,149.280
C08944=1164.520,-66.655,-43.479,179.219,5.873,149.280
C08945=1164.514,-66.405,-43.489,179.221,5.873,149.279
C08946=1164.510,-66.155,-43.500,179.223,5.873,149.278
C08947=1164.504,-65.906,-43.511,179.226,5.874,149.278
C08948=1164.498,-65.655,-43.522,179.228,5.874,149.277
C08949=1164.493,-65.406,-43.533,179.230,5.874,149.277
C08950=1164.488,-65.156,-43.543,179.233,5.875,149.276
C08951=1164.482,-64.907,-43.553,179.235,5.876,149.275
C08952=1164.478,-64.657,-43.565,179.237,5.875,149.275
C08953=1164.472,-64.408,-43.575,179.239,5.876,149.274
C08954=1164.467,-64.158,-43.586,179.242,5.876,149.274
C08955=1164.462,-63.908,-43.596,179.244,5.877,149.273
C08956=1164.456,-63.658,-43.608,179.246,5.877,149.272
C08957=1164.451,-63.409,-43.619,179.248,5.878,149.272
C08958=1164.446,-63.159,-43.629,179.251,5.878,149.271
C08959=1164.441,-62.909,-43.640,179.253,5.879,149.271
C08960=1164.436,-62.659,-43.651,179.255,5.878,149.270
C08961=1164.431,-62.410,-43.662,179.257,5.879,149.270
C08962=1164.425,-62.160,-43.672,179.260,5.880,149.269
C08963=1164.420,-61.910,-43.684,179.262,5.880,149.268
C08964=1164.414,-61.661,-43.694,179.264,5.880,149.268
C08965=1164.410,-61.411,-43.706,179.266,5.881,149.267
C08966=1164.405,-61.161,-43.716,179.269,5.881,149.266
C08967=1164.399,-60.911,-43.726,179.271,5.882,149.266
C08968=1164.394,-60.661,-43.738,179.273,5.882,149.265
C08969=1164.388,-60.413,-43.749,179.275,5.882,149.265
C08970=1164.383,-60.162,-43.760,179.278,5.883,149.264
C08971=1164.378,-59.913,-43.771,179.280,5.884,149.264
C08972=1164.373,-59.663,-43.781,179.282,5.883,149.263
C08973=1164.368,-59.413,-43.793,179.285,5.884,149.262
C08974=1164.362,-59.164,-43.803,179.287,5.884,149.262
C08975=1164.357,-58.914,-43.815,179.289,5.885,149.261
C08976=1164.352,-58.664,-43.825,179.291,5.885,149.261
C08977=1164.346,-58.415,-43.837,179.294,5.886,149.260
C08978=1164.341,-58.164,-43.847,179.296,5.886,149.259
C08979=1164.336,-57.915,-43.858,179.299,5.887,149.259
C08980=1164.331,-57.666,-43.869,179.301,5.887,149.258
C08981=1164.325,-57.415,-43.881,179.303,5.887,149.258
C08982=1164.320,-57.166,-43.892,179.305,5.888,149.257
C08983=1164.315,-56.916,-43.902,179.308,5.888,149.257
C08984=1164.310,-56.666,-43.913,179.310,5.889,149.256
C08985=1164.304,-56.417,-43.925,179.312,5.888,149.255
C08986=1164.299,-56.167,-43.935,179.315,5.889,149.255
C08987=1164.295,-55.917,-43.947,179.317,5.890,149.254
C08988=1164.289,-55.668,-43.958,179.319,5.890,149.253
C08989=1164.284,-55.418,-43.969,179.322,5.891,149.253
C08990=1164.279,-55.168,-43.980,179.324,5.891,149.252
C08991=1164.273,-54.919,-43.992,179.326,5.891,149.252
C08992=1164.268,-54.669,-44.002,179.329,5.892,149.251
C08993=1164.263,-54.419,-44.014,179.331,5.892,149.250
C08994=1164.257,-54.170,-44.025,179.333,5.892,149.250
C08995=1164.252,-53.920,-44.036,179.335,5.893,149.249
C08996=1164.248,-53.670,-44.047,179.338,5.894,149.249
C08997=1164.242,-53.421,-44.058,179.340,5.894,149.248
C08998=1164.237,-53.171,-44.070,179.342,5.895,149.248
C08999=1164.232,-52.921,-44.080,179.345,5.894,149.247
C09000=1164.226,-52.672,-44.092,179.347,5.895,149.246
C09001=1164.221,-52.422,-44.103,179.349,5.896,149.246
C09002=1164.216,-52.172,-44.114,179.352,5.896,149.245
C09003=1164.211,-51.922,-44.126,179.354,5.897,149.245
C09004=1164.205,-51.673,-44.137,179.356,5.896,149.244
C09005=1164.200,-51.423,-44.148,179.359,5.897,149.243
C09006=1164.195,-51.173,-44.160,179.361,5.898,149.243
C09007=1164.190,-50.924,-44.170,179.363,5.898,149.242
C09008=1164.184,-50.674,-44.182,179.366,5.899,149.241
C09009=1164.179,-50.403,-44.194,179.368,5.900,149.241
C09010=1164.173,-50.133,-44.207,179.371,5.900,149.240
C09011=1164.167,-49.862,-44.219,179.374,5.900,149.240
C09012=1164.162,-49.592,-44.231,179.376,5.900,149.239
C09013=1164.156,-49.342,-44.242,179.378,5.901,149.238
C09014=1164.152,-49.093,-44.253,179.380,5.901,149.238
C09015=1164.146,-48.843,-44.265,179.383,5.902,149.237
C09016=1164.141,-48.593,-44.277,179.385,5.902,149.236
C09017=1164.135,-48.344,-44.288,179.388,5.903,149.236
C09018=1164.131,-48.094,-44.299,179.390,5.903,149.235
C09019=1164.125,-47.844,-44.311,179.392,5.904,149.235
C09020=1164.120,-47.594,-44.322,179.394,5.904,149.234
C09021=1164.114,-47.345,-44.333,179.397,5.905,149.234
C09022=1164.110,-47.095,-44.345,179.399,5.905,149.233
C09023=1164.104,-46.845,-44.356,179.401,5.905,149.232
C09024=1164.099,-46.596,-44.368,179.404,5.906,149.232
C09025=1164.094,-46.346,-44.380,179.406,5.906,149.231
C09026=1164.089,-46.097,-44.391,179.408,5.907,149.231
C09027=1164.083,-45.847,-44.402,179.411,5.907,149.230
C09028=1164.079,-45.597,-44.414,179.413,5.908,149.229
C09029=1164.073,-45.347,-44.426,179.415,5.908,149.229
C09030=1164.068,-45.098,-44.437,179.418,5.909,149.228
C09031=1164.062,-44.848,-44.448,179.420,5.909,149.228
C09032=1164.058,-44.599,-44.460,179.422,5.910,149.227
C09033=1164.052,-44.349,-44.472,179.425,5.910,149.226
C09034=1164.047,-44.099,-44.484,179.428,5.911,149.226
C09035=1164.042,-43.849,-44.495,179.429,5.911,149.225
C09036=1164.037,-43.599,-44.507,179.432,5.911,149.224
C09037=1164.031,-43.350,-44.518,179.434,5.912,149.224
C09038=1164.026,-43.101,-44.530,179.437,5.912,149.223
C09039=1164.021,-42.851,-44.541,179.439,5.913,149.223
C09040=1164.016,-42.601,-44.553,179.442,5.913,149.222
C09041=1164.011,-42.351,-44.565,179.444,5.914,149.222
C09042=1164.006,-42.101,-44.576,179.446,5.914,149.221
C09043=1164.000,-41.852,-44.587,179.448,5.915,149.220
C09044=1163.995,-41.603,-44.599,179.451,5.915,149.220
C09045=1163.990,-41.353,-44.611,179.453,5.916,149.219
C09046=1163.984,-41.103,-44.622,179.456,5.916,149.219
C09047=1163.980,-40.853,-44.634,179.458,5.917,149.218
C09048=1163.974,-40.603,-44.646,179.460,5.918,149.217
C09049=1163.969,-40.353,-44.657,179.463,5.917,149.217
C09050=1163.964,-40.104,-44.669,179.465,5.918,149.216
C09051=1163.958,-39.855,-44.681,179.467,5.918,149.216
C09052=1163.953,-39.605,-44.693,179.470,5.919,149.215
C09053=1163.948,-39.355,-44.704,179.472,5.920,149.214
C09054=1163.943,-39.105,-44.716,179.474,5.920,149.214
C09055=1163.937,-38.855,-44.728,179.477,5.921,149.213
C09056=1163.933,-38.606,-44.739,179.479,5.920,149.213
C09057=1163.927,-38.356,-44.751,179.481,5.921,149.212
C09058=1163.922,-38.107,-44.764,179.484,5.922,149.211
C09059=1163.917,-37.857,-44.775,179.486,5.923,149.211
C09060=1163.911,-37.608,-44.787,179.489,5.923,149.210
C09061=1163.906,-37.358,-44.798,179.491,5.924,149.210
C09062=1163.900,-37.108,-44.810,179.494,5.924,149.209
C09063=1163.896,-36.859,-44.822,179.496,5.925,149.209
C09064=1163.891,-36.609,-44.834,179.498,5.925,149.208
C09065=1163.885,-36.359,-44.846,179.501,5.925,149.207
C09066=1163.881,-36.109,-44.857,179.503,5.926,149.207
C09067=1163.875,-35.860,-44.870,179.505,5.926,149.206
C09068=1163.870,-35.610,-44.882,179.508,5.927,149.205
C09069=1163.865,-35.360,-44.894,179.510,5.927,149.205
C09070=1163.859,-35.110,-44.906,179.512,5.928,149.204
C09071=1163.855,-34.861,-44.918,179.515,5.929,149.204
C09072=1163.849,-34.611,-44.930,179.517,5.929,149.203
C09073=1163.844,-34.361,-44.941,179.519,5.929,149.202
C09074=1163.839,-34.112,-44.954,179.522,5.930,149.202
C09075=1163.834,-33.862,-44.965,179.524,5.930,149.201
C09076=1163.829,-33.612,-44.977,179.527,5.931,149.201
C09077=1163.823,-33.363,-44.990,179.529,5.932,149.200
C09078=1163.818,-33.113,-45.002,179.532,5.932,149.199
C09079=1163.813,-32.863,-45.014,179.534,5.933,149.199
C09080=1163.808,-32.614,-45.026,179.537,5.933,149.198
C09081=1163.803,-32.364,-45.037,179.538,5.933,149.198
C09082=1163.797,-32.114,-45.049,179.541,5.934,149.197
C09083=1163.792,-31.865,-45.062,179.543,5.934,149.196
C09084=1163.787,-31.615,-45.074,179.546,5.935,149.196
C09085=1163.781,-31.365,-45.086,179.548,5.935,149.195
C09086=1163.777,-31.116,-45.098,179.551,5.936,149.195
C09087=1163.772,-30.866,-45.110,179.553,5.937,149.194
C09088=1163.766,-30.617,-45.122,179.555,5.937,149.194
C09089=1163.761,-30.367,-45.134,179.558,5.938,149.193
C09090=1163.756,-30.117,-45.146,179.560,5.939,149.192
C09091=1163.750,-29.868,-45.159,179.563,5.939,149.192
C09092=1163.745,-29.618,-45.170,179.565,5.939,149.191
C09093=1163.741,-29.369,-45.182,179.567,5.940,149.190
C09094=1163.735,-29.119,-45.194,179.570,5.940,149.190
C09095=1163.730,-28.870,-45.207,179.572,5.941,149.189
C09096=1163.725,-28.620,-45.219,179.575,5.941,149.189
C09097=1163.720,-28.370,-45.231,179.577,5.942,149.188
C09098=1163.714,-28.120,-45.243,179.579,5.942,149.187
C09099=1163.709,-27.871,-45.256,179.582,5.943,149.187
C09100=1163.704,-27.621,-45.268,179.584,5.944,149.186
C09101=1163.698,-27.372,-45.280,179.587,5.944,149.186
C09102=1163.693,-27.122,-45.292,179.589,5.945,149.185
C09103=1163.688,-26.873,-45.305,179.592,5.945,149.184
C09104=1163.683,-26.622,-45.317,179.594,5.946,149.184
C09105=1163.679,-26.373,-45.329,179.596,5.946,149.183
C09106=1163.673,-26.123,-45.341,179.598,5.947,149.183
C09107=1163.668,-25.874,-45.354,179.601,5.947,149.182
C09108=1163.663,-25.624,-45.366,179.604,5.947,149.181
C09109=1163.658,-25.374,-45.378,179.606,5.948,149.181
C09110=1163.652,-25.125,-45.391,179.608,5.949,149.180
C09111=1163.647,-24.875,-45.403,179.611,5.949,149.180
C09112=1163.642,-24.626,-45.415,179.613,5.950,149.179
C09113=1163.636,-24.355,-45.429,179.616,5.950,149.178
C09114=1163.631,-24.085,-45.442,179.618,5.951,149.178
C09115=1163.625,-23.816,-45.455,179.621,5.952,149.177
C09116=1163.620,-23.546,-45.469,179.623,5.952,149.176
C09117=1163.615,-23.297,-45.481,179.626,5.952,149.176
C09118=1163.609,-23.047,-45.494,179.628,5.953,149.175
C09119=1163.604,-22.797,-45.506,179.631,5.954,149.175
C09120=1163.598,-22.548,-45.519,179.633,5.955,149.174
C09121=1163.594,-22.297,-45.531,179.636,5.955,149.173
C09122=1163.588,-22.048,-45.544,179.638,5.956,149.173
C09123=1163.583,-21.799,-45.556,179.641,5.956,149.172
C09124=1163.578,-21.549,-45.568,179.643,5.957,149.172
C09125=1163.573,-21.299,-45.581,179.645,5.957,149.171
C09126=1163.568,-21.050,-45.594,179.648,5.958,149.170
C09127=1163.563,-20.799,-45.606,179.650,5.959,149.170
C09128=1163.558,-20.550,-45.618,179.653,5.959,149.169
C09129=1163.553,-20.301,-45.631,179.655,5.960,149.169
C09130=1163.547,-20.051,-45.644,179.658,5.960,149.168
C09131=1163.542,-19.802,-45.655,179.660,5.961,149.168
C09132=1163.536,-19.552,-45.669,179.663,5.962,149.167
C09133=1163.532,-19.302,-45.682,179.665,5.962,149.166
C09134=1163.527,-19.053,-45.694,179.667,5.963,149.166
C09135=1163.521,-18.803,-45.706,179.670,5.963,149.165
C09136=1163.516,-18.553,-45.719,179.672,5.964,149.165
C09137=1163.511,-18.304,-45.731,179.675,5.965,149.164
C09138=1163.506,-18.054,-45.744,179.677,5.965,149.163
C09139=1163.500,-17.804,-45.758,179.680,5.966,149.163
C09140=1163.495,-17.555,-45.770,179.682,5.965,149.162
C09141=1163.490,-17.305,-45.782,179.684,5.966,149.162
C09142=1163.485,-17.055,-45.795,179.687,5.967,149.161
C09143=1163.480,-16.806,-45.808,179.689,5.968,149.160
C09144=1163.475,-16.556,-45.820,179.692,5.968,149.160
C09145=1163.469,-16.307,-45.833,179.694,5.969,149.159
C09146=1163.464,-16.057,-45.846,179.696,5.969,149.159
C09147=1163.460,-15.807,-45.859,179.699,5.970,149.158
C09148=1163.454,-15.558,-45.871,179.701,5.970,149.157
C09149=1163.449,-15.308,-45.883,179.704,5.971,149.157
C09150=1163.443,-15.059,-45.897,179.706,5.972,149.156
C09151=1163.439,-14.809,-45.910,179.709,5.972,149.156
C09152=1163.434,-14.559,-45.922,179.711,5.973,149.155
C09153=1163.428,-14.310,-45.935,179.714,5.973,149.154
C09154=1163.424,-14.060,-45.948,179.716,5.974,149.154
C09155=1163.418,-13.810,-45.961,179.718,5.975,149.153
